LIN {X 0,Y 495.75,Z 552.238,A -85,B 0,C 180,E1 16037.936,E2 16037.936} C_VEL
LIN {X 0,Y 490.414,Z 542.078,A -85,B 0,C 180,E1 16035.4,E2 16035.4} C_VEL
LIN {X 0,Y 486.83,Z 535.501,A -85,B 0,C 180,E1 16033.42,E2 16033.42} C_VEL
LIN {X 0,Y 483.427,Z 530.223,A -85,B 0,C 180,E1 16031.272,E2 16031.272} C_VEL
LIN {X 0,Y 481.027,Z 526.46,A -85,B 0,C 180,E1 16029.452,E2 16029.452} C_VEL
LIN {X 0,Y 478.245,Z 521.895,A -85,B 0,C 180,E1 16026.724,E2 16026.724} C_VEL
LIN {X 0,Y 475.904,Z 518.407,A -85,B 0,C 180,E1 16023.011,E2 16023.011} C_VEL
LIN {X 0,Y 475.553,Z 516.68,A -85,B 0,C 180,E1 16021.446,E2 16021.446} C_VEL
LIN {X 0,Y 475.613,Z 516.934,A -85,B 0,C 180,E1 16017.711,E2 16017.711} C_VEL
LIN {X 0,Y 477.41,Z 521.143,A -85,B 0,C 180,E1 16013.748,E2 16013.748} C_VEL
LIN {X 0,Y 478.53,Z 522.413,A -85,B 0,C 180,E1 16012.436,E2 16012.436} C_VEL
LIN {X 0,Y 481.805,Z 527.661,A -85,B 0,C 180,E1 16009.417,E2 16009.417} C_VEL
LIN {X 0,Y 485.153,Z 532.978,A -85,B 0,C 180,E1 16007.078,E2 16007.078} C_VEL
LIN {X 0,Y 488.531,Z 538.287,A -85,B 0,C 180,E1 16005.116,E2 16005.116} C_VEL
LIN {X 0,Y 494.078,Z 547.334,A -85,B 0,C 180,E1 16002.389,E2 16002.389} C_VEL
LIN {X 0,Y 495.655,Z 550.313,A -85,B 0,C 180,E1 16001.678,E2 16001.678} C_VEL
LIN {X 0,Y 477.005,Z 773.14,A -85,B 0,C 180,E1 15998.26,E2 15998.26} C_VEL
LIN {X 0,Y 473.208,Z 814.507,A -85,B 0,C 180,E1 15997.599,E2 15997.599} C_VEL
LIN {X 0,Y 469.106,Z 841.171,A -85,B 0,C 180,E1 15997.058,E2 15997.058} C_VEL
LIN {X 0,Y 464.96,Z 862.529,A -85,B 0,C 180,E1 15996.503,E2 15996.503} C_VEL
LIN {X 0,Y 460.196,Z 883.041,A -85,B 0,C 180,E1 15995.856,E2 15995.856} C_VEL
LIN {X 0,Y 454.375,Z 904.584,A -85,B 0,C 180,E1 15995.041,E2 15995.041} C_VEL
LIN {X 0,Y 446.157,Z 930.766,A -85,B 0,C 180,E1 15993.836,E2 15993.836} C_VEL
LIN {X 0,Y 438.115,Z 952.919,A -85,B 0,C 180,E1 15992.594,E2 15992.594} C_VEL
LIN {X 0,Y 430.587,Z 971.671,A -85,B 0,C 180,E1 15991.371,E2 15991.371} C_VEL
LIN {X 0,Y 422.617,Z 989.978,A -85,B 0,C 180,E1 15989.986,E2 15989.986} C_VEL
LIN {X 0,Y 414.059,Z 1008.193,A -85,B 0,C 180,E1 15988.397,E2 15988.397} C_VEL
LIN {X 0,Y 402.823,Z 1030.327,A -85,B 0,C 180,E1 15986.126,E2 15986.126} C_VEL
LIN {X 0,Y 392.874,Z 1048.447,A -85,B 0,C 180,E1 15983.904,E2 15983.904} C_VEL
LIN {X 0,Y 384.294,Z 1063.355,A -85,B 0,C 180,E1 15981.789,E2 15981.789} C_VEL
LIN {X 0,Y 375.957,Z 1077.309,A -85,B 0,C 180,E1 15979.518,E2 15979.518} C_VEL
LIN {X 0,Y 367.251,Z 1091.49,A -85,B 0,C 180,E1 15976.856,E2 15976.856} C_VEL
LIN {X 0,Y 357.211,Z 1107.595,A -85,B 0,C 180,E1 15973.296,E2 15973.296} C_VEL
LIN {X 0,Y 348.718,Z 1120.908,A -85,B 0,C 180,E1 15969.747,E2 15969.747} C_VEL
LIN {X 0,Y 342.021,Z 1131.618,A -85,B 0,C 180,E1 15966.402,E2 15966.402} C_VEL
LIN {X 0,Y 336.338,Z 1141.067,A -85,B 0,C 180,E1 15962.957,E2 15962.957} C_VEL
LIN {X 0,Y 330.571,Z 1151.31,A -85,B 0,C 180,E1 15958.548,E2 15958.548} C_VEL
LIN {X 0,Y 326.088,Z 1159.977,A -85,B 0,C 180,E1 15953.875,E2 15953.875} C_VEL
LIN {X 0,Y 323.408,Z 1166.015,A -85,B 0,C 180,E1 15949.882,E2 15949.882} C_VEL
LIN {X 0,Y 321.713,Z 1170.693,A -85,B 0,C 180,E1 15946.058,E2 15946.058} C_VEL
LIN {X 0,Y 320.731,Z 1174.188,A -85,B 0,C 180,E1 15942.422,E2 15942.422} C_VEL
LIN {X 0,Y 320.245,Z 1176.775,A -85,B 0,C 180,E1 15938.8,E2 15938.8} C_VEL
LIN {X 0,Y 320.04,Z 1178.413,A -85,B 0,C 180,E1 15935.378,E2 15935.378} C_VEL
LIN {X 0,Y 319.982,Z 1179.268,A -85,B 0,C 180,E1 15931.97,E2 15931.97} C_VEL
LIN {X 0,Y 319.983,Z 1179.345,A -85,B 0,C 180,E1 15928.568,E2 15928.568} C_VEL
LIN {X 0,Y 320.024,Z 1178.581,A -85,B 0,C 180,E1 15924.981,E2 15924.981} C_VEL
LIN {X 0,Y 320.225,Z 1176.946,A -85,B 0,C 180,E1 15921.38,E2 15921.38} C_VEL
LIN {X 0,Y 320.681,Z 1174.428,A -85,B 0,C 180,E1 15917.759,E2 15917.759} C_VEL
LIN {X 0,Y 321.622,Z 1171.003,A -85,B 0,C 180,E1 15914.123,E2 15914.123} C_VEL
LIN {X 0,Y 323.269,Z 1166.396,A -85,B 0,C 180,E1 15910.298,E2 15910.298} C_VEL
LIN {X 0,Y 325.73,Z 1160.725,A -85,B 0,C 180,E1 15906.481,E2 15906.481} C_VEL
LIN {X 0,Y 329.298,Z 1153.603,A -85,B 0,C 180,E1 15902.515,E2 15902.515} C_VEL
LIN {X 0,Y 335.203,Z 1143.09,A -85,B 0,C 180,E1 15897.729,E2 15897.729} C_VEL
LIN {X 0,Y 341.588,Z 1132.376,A -85,B 0,C 180,E1 15893.753,E2 15893.753} C_VEL
LIN {X 0,Y 348.208,Z 1121.753,A -85,B 0,C 180,E1 15890.398,E2 15890.398} C_VEL
LIN {X 0,Y 355.813,Z 1109.777,A -85,B 0,C 180,E1 15887.154,E2 15887.154} C_VEL
LIN {X 0,Y 366.624,Z 1092.626,A -85,B 0,C 180,E1 15883.268,E2 15883.268} C_VEL
LIN {X 0,Y 372.671,Z 1082.974,A -85,B 0,C 180,E1 15881.378,E2 15881.378} C_VEL
LIN {X 0,Y 374.707,Z 1078.514,A -85,B 0,C 180,E1 15880.457,E2 15880.457} C_VEL
LIN {X 0,Y 377.403,Z 1067.82,A -85,B 0,C 180,E1 15877.896,E2 15877.896} C_VEL
LIN {X 0,Y 379.662,Z 1063.03,A -85,B 0,C 180,E1 15877.03,E2 15877.03} C_VEL
LIN {X 0,Y 390.229,Z 1045.195,A -85,B 0,C 180,E1 15874.537,E2 15874.537} C_VEL
LIN {X 0,Y 401.817,Z 1024.144,A -85,B 0,C 180,E1 15872.083,E2 15872.083} C_VEL
LIN {X 0,Y 411.116,Z 1006.054,A -85,B 0,C 180,E1 15870.302,E2 15870.302} C_VEL
LIN {X 0,Y 419.413,Z 988.742,A -85,B 0,C 180,E1 15868.825,E2 15868.825} C_VEL
LIN {X 0,Y 427.593,Z 970.262,A -85,B 0,C 180,E1 15867.452,E2 15867.452} C_VEL
LIN {X 0,Y 437.088,Z 946.84,A -85,B 0,C 180,E1 15865.973,E2 15865.973} C_VEL
LIN {X 0,Y 445.714,Z 922.226,A -85,B 0,C 180,E1 15864.698,E2 15864.698} C_VEL
LIN {X 0,Y 451.949,Z 902.144,A -85,B 0,C 180,E1 15863.824,E2 15863.824} C_VEL
LIN {X 0,Y 457.53,Z 881.65,A -85,B 0,C 180,E1 15863.07,E2 15863.07} C_VEL
LIN {X 0,Y 462.528,Z 860.189,A -85,B 0,C 180,E1 15862.411,E2 15862.411} C_VEL
LIN {X 0,Y 467.655,Z 833.351,A -85,B 0,C 180,E1 15861.757,E2 15861.757} C_VEL
LIN {X 0,Y 471.236,Z 806.582,A -85,B 0,C 180,E1 15861.267,E2 15861.267} C_VEL
LIN {X 0,Y 483.431,Z 664.825,A -85,B 0,C 180,E1 15859.081,E2 15859.081} C_VEL
LIN {X 0,Y 492.923,Z 555.55,A -85,B 0,C 180,E1 15857.416,E2 15857.416} C_VEL
LIN {X 0,Y 487.652,Z 546.708,A -85,B 0,C 180,E1 15854.79,E2 15854.79} C_VEL
LIN {X 0,Y 484.383,Z 541.518,A -85,B 0,C 180,E1 15852.882,E2 15852.882} C_VEL
LIN {X 0,Y 482.213,Z 538.052,A -85,B 0,C 180,E1 15851.421,E2 15851.421} C_VEL
LIN {X 0,Y 479.901,Z 534.242,A -85,B 0,C 180,E1 15849.595,E2 15849.595} C_VEL
LIN {X 0,Y 477.233,Z 529.795,A -85,B 0,C 180,E1 15846.859,E2 15846.859} C_VEL
LIN {X 0,Y 474.881,Z 525.658,A -85,B 0,C 180,E1 15842.414,E2 15842.414} C_VEL
LIN {X 0,Y 474.762,Z 524.669,A -85,B 0,C 180,E1 15841.448,E2 15841.448} C_VEL
LIN {X 0,Y 474.801,Z 524.83,A -85,B 0,C 180,E1 15838.673,E2 15838.673} C_VEL
LIN {X 0,Y 476.414,Z 529.01,A -85,B 0,C 180,E1 15834.581,E2 15834.581} C_VEL
LIN {X 0,Y 477.632,Z 530.406,A -85,B 0,C 180,E1 15833.086,E2 15833.086} C_VEL
LIN {X 0,Y 480.894,Z 535.8,A -85,B 0,C 180,E1 15830.002,E2 15830.002} C_VEL
LIN {X 0,Y 483.748,Z 540.41,A -85,B 0,C 180,E1 15827.95,E2 15827.95} C_VEL
LIN {X 0,Y 486.694,Z 545.279,A -85,B 0,C 180,E1 15826.152,E2 15826.152} C_VEL
LIN {X 0,Y 492.309,Z 556.092,A -85,B 0,C 180,E1 15823.207,E2 15823.207} C_VEL
LIN {X 0,Y 492.992,Z 557.773,A -85,B 0,C 180,E1 15822.869,E2 15822.869} C_VEL
LIN {X 0,Y 474.136,Z 778.593,A -85,B 0,C 180,E1 15819.49,E2 15819.49} C_VEL
LIN {X 0,Y 469.97,Z 824.297,A -85,B 0,C 180,E1 15818.766,E2 15818.766} C_VEL
LIN {X 0,Y 465.648,Z 852.231,A -85,B 0,C 180,E1 15818.23,E2 15818.23} C_VEL
LIN {X 0,Y 461.221,Z 874.106,A -85,B 0,C 180,E1 15817.714,E2 15817.714} C_VEL
LIN {X 0,Y 456.149,Z 895.17,A -85,B 0,C 180,E1 15817.097,E2 15817.097} C_VEL
LIN {X 0,Y 449.874,Z 917.56,A -85,B 0,C 180,E1 15816.302,E2 15816.302} C_VEL
LIN {X 0,Y 440.941,Z 944.901,A -85,B 0,C 180,E1 15815.096,E2 15815.096} C_VEL
LIN {X 0,Y 432.943,Z 966.301,A -85,B 0,C 180,E1 15813.945,E2 15813.945} C_VEL
LIN {X 0,Y 425.158,Z 985.312,A -85,B 0,C 180,E1 15812.742,E2 15812.742} C_VEL
LIN {X 0,Y 416.857,Z 1003.907,A -85,B 0,C 180,E1 15811.387,E2 15811.387} C_VEL
LIN {X 0,Y 406.65,Z 1025.184,A -85,B 0,C 180,E1 15809.567,E2 15809.567} C_VEL
LIN {X 0,Y 394.948,Z 1047.489,A -85,B 0,C 180,E1 15807.268,E2 15807.268} C_VEL
LIN {X 0,Y 385.523,Z 1064.419,A -85,B 0,C 180,E1 15805.208,E2 15805.208} C_VEL
LIN {X 0,Y 376.324,Z 1080.251,A -85,B 0,C 180,E1 15802.977,E2 15802.977} C_VEL
LIN {X 0,Y 366.484,Z 1096.63,A -85,B 0,C 180,E1 15800.297,E2 15800.297} C_VEL
LIN {X 0,Y 355.351,Z 1114.595,A -85,B 0,C 180,E1 15796.782,E2 15796.782} C_VEL
LIN {X 0,Y 346.694,Z 1128.363,A -85,B 0,C 180,E1 15793.572,E2 15793.572} C_VEL
LIN {X 0,Y 339.406,Z 1140.072,A -85,B 0,C 180,E1 15790.398,E2 15790.398} C_VEL
LIN {X 0,Y 332.394,Z 1151.594,A -85,B 0,C 180,E1 15786.77,E2 15786.77} C_VEL
LIN {X 0,Y 324.831,Z 1164.761,A -85,B 0,C 180,E1 15781.759,E2 15781.759} C_VEL
LIN {X 0,Y 320.263,Z 1173.478,A -85,B 0,C 180,E1 15777.722,E2 15777.722} C_VEL
LIN {X 0,Y 316.98,Z 1180.584,A -85,B 0,C 180,E1 15773.813,E2 15773.813} C_VEL
LIN {X 0,Y 314.614,Z 1186.622,A -85,B 0,C 180,E1 15769.824,E2 15769.824} C_VEL
LIN {X 0,Y 312.967,Z 1192.261,A -85,B 0,C 180,E1 15765.187,E2 15765.187} C_VEL
LIN {X 0,Y 312.171,Z 1196.482,A -85,B 0,C 180,E1 15760.333,E2 15760.333} C_VEL
LIN {X 0,Y 311.987,Z 1198.799,A -85,B 0,C 180,E1 15756.256,E2 15756.256} C_VEL
LIN {X 0,Y 311.979,Z 1199.933,A -85,B 0,C 180,E1 15752.572,E2 15752.572} C_VEL
LIN {X 0,Y 311.983,Z 1200.121,A -85,B 0,C 180,E1 15748.898,E2 15748.898} C_VEL
LIN {X 0,Y 311.974,Z 1199.365,A -85,B 0,C 180,E1 15745.22,E2 15745.22} C_VEL
LIN {X 0,Y 312.051,Z 1197.662,A -85,B 0,C 180,E1 15741.524,E2 15741.524} C_VEL
LIN {X 0,Y 312.398,Z 1194.842,A -85,B 0,C 180,E1 15737.617,E2 15737.617} C_VEL
LIN {X 0,Y 313.276,Z 1190.964,A -85,B 0,C 180,E1 15733.688,E2 15733.688} C_VEL
LIN {X 0,Y 314.826,Z 1186.005,A -85,B 0,C 180,E1 15729.747,E2 15729.747} C_VEL
LIN {X 0,Y 317.113,Z 1180.25,A -85,B 0,C 180,E1 15726,E2 15726} C_VEL
LIN {X 0,Y 320.564,Z 1172.85,A -85,B 0,C 180,E1 15721.973,E2 15721.973} C_VEL
LIN {X 0,Y 326.29,Z 1162.177,A -85,B 0,C 180,E1 15717.154,E2 15717.154} C_VEL
LIN {X 0,Y 333.014,Z 1150.506,A -85,B 0,C 180,E1 15712.88,E2 15712.88} C_VEL
LIN {X 0,Y 339.761,Z 1139.443,A -85,B 0,C 180,E1 15709.431,E2 15709.431} C_VEL
LIN {X 0,Y 347.501,Z 1127.012,A -85,B 0,C 180,E1 15706.098,E2 15706.098} C_VEL
LIN {X 0,Y 358.082,Z 1110.175,A -85,B 0,C 180,E1 15702.296,E2 15702.296} C_VEL
LIN {X 0,Y 368.02,Z 1093.965,A -85,B 0,C 180,E1 15699.258,E2 15699.258} C_VEL
LIN {X 0,Y 377.147,Z 1078.74,A -85,B 0,C 180,E1 15696.81,E2 15696.81} C_VEL
LIN {X 0,Y 386.604,Z 1062.403,A -85,B 0,C 180,E1 15694.541,E2 15694.541} C_VEL
LIN {X 0,Y 398.513,Z 1040.77,A -85,B 0,C 180,E1 15692.002,E2 15692.002} C_VEL
LIN {X 0,Y 408.806,Z 1020.52,A -85,B 0,C 180,E1 15690.025,E2 15690.025} C_VEL
LIN {X 0,Y 417.516,Z 1002.219,A -85,B 0,C 180,E1 15688.492,E2 15688.492} C_VEL
LIN {X 0,Y 425.839,Z 983.449,A -85,B 0,C 180,E1 15687.142,E2 15687.142} C_VEL
LIN {X 0,Y 434.731,Z 961.518,A -85,B 0,C 180,E1 15685.786,E2 15685.786} C_VEL
LIN {X 0,Y 443.915,Z 935.872,A -85,B 0,C 180,E1 15684.485,E2 15684.485} C_VEL
LIN {X 0,Y 450.606,Z 914.601,A -85,B 0,C 180,E1 15683.593,E2 15683.593} C_VEL
LIN {X 0,Y 456.321,Z 893.984,A -85,B 0,C 180,E1 15682.873,E2 15682.873} C_VEL
LIN {X 0,Y 461.332,Z 872.995,A -85,B 0,C 180,E1 15682.264,E2 15682.264} C_VEL
LIN {X 0,Y 466.121,Z 848.981,A -85,B 0,C 180,E1 15681.709,E2 15681.709} C_VEL
LIN {X 0,Y 470.294,Z 819.745,A -85,B 0,C 180,E1 15681.166,E2 15681.166} C_VEL
LIN {X 0,Y 476.185,Z 752.192,A -85,B 0,C 180,E1 15680.11,E2 15680.11} C_VEL
LIN {X 0,Y 492.837,Z 557.39,A -85,B 0,C 180,E1 15677.124,E2 15677.124} C_VEL
LIN {X 0,Y 487.943,Z 547.91,A -85,B 0,C 180,E1 15674.66,E2 15674.66} C_VEL
LIN {X 0,Y 485.144,Z 542.775,A -85,B 0,C 180,E1 15673.043,E2 15673.043} C_VEL
LIN {X 0,Y 482.105,Z 537.911,A -85,B 0,C 180,E1 15671.061,E2 15671.061} C_VEL
LIN {X 0,Y 479.904,Z 534.344,A -85,B 0,C 180,E1 15669.353,E2 15669.353} C_VEL
LIN {X 0,Y 477.055,Z 529.687,A -85,B 0,C 180,E1 15666.499,E2 15666.499} C_VEL
LIN {X 0,Y 474.846,Z 526.136,A -85,B 0,C 180,E1 15662.776,E2 15662.776} C_VEL
LIN {X 0,Y 474.55,Z 524.614,A -85,B 0,C 180,E1 15661.328,E2 15661.328} C_VEL
LIN {X 0,Y 474.611,Z 524.819,A -85,B 0,C 180,E1 15657.827,E2 15657.827} C_VEL
LIN {X 0,Y 476.436,Z 529.122,A -85,B 0,C 180,E1 15653.735,E2 15653.735} C_VEL
LIN {X 0,Y 477.439,Z 530.341,A -85,B 0,C 180,E1 15652.539,E2 15652.539} C_VEL
LIN {X 0,Y 480.592,Z 535.493,A -85,B 0,C 180,E1 15649.572,E2 15649.572} C_VEL
LIN {X 0,Y 483.792,Z 540.671,A -85,B 0,C 180,E1 15647.287,E2 15647.287} C_VEL
LIN {X 0,Y 487.114,Z 545.999,A -85,B 0,C 180,E1 15645.315,E2 15645.315} C_VEL
LIN {X 0,Y 492.64,Z 555.185,A -85,B 0,C 180,E1 15642.549,E2 15642.549} C_VEL
LIN {X 0,Y 492.74,Z 555.792,A -85,B 0,C 180,E1 15642.482,E2 15642.482} C_VEL
LIN {X 0,Y 473.681,Z 778.427,A -85,B 0,C 180,E1 15639.082,E2 15639.082} C_VEL
LIN {X 0,Y 470.001,Z 816.245,A -85,B 0,C 180,E1 15638.474,E2 15638.474} C_VEL
LIN {X 0,Y 465.993,Z 841.708,A -85,B 0,C 180,E1 15637.959,E2 15637.959} C_VEL
LIN {X 0,Y 461.747,Z 863.128,A -85,B 0,C 180,E1 15637.408,E2 15637.408} C_VEL
LIN {X 0,Y 456.779,Z 884.051,A -85,B 0,C 180,E1 15636.751,E2 15636.751} C_VEL
LIN {X 0,Y 450.303,Z 907.411,A -85,B 0,C 180,E1 15635.865,E2 15635.865} C_VEL
LIN {X 0,Y 441.922,Z 933.032,A -85,B 0,C 180,E1 15634.672,E2 15634.672} C_VEL
LIN {X 0,Y 434.435,Z 953.191,A -85,B 0,C 180,E1 15633.545,E2 15633.545} C_VEL
LIN {X 0,Y 426.746,Z 971.943,A -85,B 0,C 180,E1 15632.331,E2 15632.331} C_VEL
LIN {X 0,Y 418.595,Z 990.251,A -85,B 0,C 180,E1 15630.954,E2 15630.954} C_VEL
LIN {X 0,Y 410.011,Z 1008.079,A -85,B 0,C 180,E1 15629.41,E2 15629.41} C_VEL
LIN {X 0,Y 398.607,Z 1030.052,A -85,B 0,C 180,E1 15627.172,E2 15627.172} C_VEL
LIN {X 0,Y 388.064,Z 1048.722,A -85,B 0,C 180,E1 15624.89,E2 15624.89} C_VEL
LIN {X 0,Y 379.22,Z 1063.631,A -85,B 0,C 180,E1 15622.774,E2 15622.774} C_VEL
LIN {X 0,Y 370.328,Z 1078.042,A -85,B 0,C 180,E1 15620.416,E2 15620.416} C_VEL
LIN {X 0,Y 360.658,Z 1093.281,A -85,B 0,C 180,E1 15617.513,E2 15617.513} C_VEL
LIN {X 0,Y 349.663,Z 1110.098,A -85,B 0,C 180,E1 15613.658,E2 15613.658} C_VEL
LIN {X 0,Y 341.598,Z 1122.307,A -85,B 0,C 180,E1 15610.306,E2 15610.306} C_VEL
LIN {X 0,Y 334.698,Z 1132.9,A -85,B 0,C 180,E1 15606.902,E2 15606.902} C_VEL
LIN {X 0,Y 327.717,Z 1144.13,A -85,B 0,C 180,E1 15602.637,E2 15602.637} C_VEL
LIN {X 0,Y 321.842,Z 1154.033,A -85,B 0,C 180,E1 15597.976,E2 15597.976} C_VEL
LIN {X 0,Y 318.242,Z 1160.836,A -85,B 0,C 180,E1 15594.107,E2 15594.107} C_VEL
LIN {X 0,Y 315.58,Z 1166.532,A -85,B 0,C 180,E1 15590.203,E2 15590.203} C_VEL
LIN {X 0,Y 313.8,Z 1171.161,A -85,B 0,C 180,E1 15586.284,E2 15586.284} C_VEL
LIN {X 0,Y 312.73,Z 1174.763,A -85,B 0,C 180,E1 15582.369,E2 15582.369} C_VEL
LIN {X 0,Y 312.206,Z 1177.493,A -85,B 0,C 180,E1 15578.259,E2 15578.259} C_VEL
LIN {X 0,Y 312.01,Z 1179.329,A -85,B 0,C 180,E1 15573.675,E2 15573.675} C_VEL
LIN {X 0,Y 311.98,Z 1179.696,A -85,B 0,C 180,E1 15569.265,E2 15569.265} C_VEL
LIN {X 0,Y 312.026,Z 1178.975,A -85,B 0,C 180,E1 15565.221,E2 15565.221} C_VEL
LIN {X 0,Y 312.237,Z 1177.32,A -85,B 0,C 180,E1 15561.344,E2 15561.344} C_VEL
LIN {X 0,Y 312.753,Z 1174.694,A -85,B 0,C 180,E1 15557.444,E2 15557.444} C_VEL
LIN {X 0,Y 313.767,Z 1171.27,A -85,B 0,C 180,E1 15553.715,E2 15553.715} C_VEL
LIN {X 0,Y 315.537,Z 1166.665,A -85,B 0,C 180,E1 15549.794,E2 15549.794} C_VEL
LIN {X 0,Y 318.173,Z 1160.995,A -85,B 0,C 180,E1 15545.888,E2 15545.888} C_VEL
LIN {X 0,Y 321.955,Z 1153.874,A -85,B 0,C 180,E1 15541.833,E2 15541.833} C_VEL
LIN {X 0,Y 328.29,Z 1143.195,A -85,B 0,C 180,E1 15536.886,E2 15536.886} C_VEL
LIN {X 0,Y 334.888,Z 1132.649,A -85,B 0,C 180,E1 15532.908,E2 15532.908} C_VEL
LIN {X 0,Y 341.823,Z 1122.024,A -85,B 0,C 180,E1 15529.506,E2 15529.506} C_VEL
LIN {X 0,Y 349.747,Z 1110.049,A -85,B 0,C 180,E1 15526.225,E2 15526.225} C_VEL
LIN {X 0,Y 360.963,Z 1092.897,A -85,B 0,C 180,E1 15522.304,E2 15522.304} C_VEL
LIN {X 0,Y 369.922,Z 1078.822,A -85,B 0,C 180,E1 15519.617,E2 15519.617} C_VEL
LIN {X 0,Y 379.214,Z 1063.772,A -85,B 0,C 180,E1 15517.144,E2 15517.144} C_VEL
LIN {X 0,Y 379.662,Z 1063.03,A -85,B 0,C 180,E1 15517.03,E2 15517.03} C_VEL
LIN {X 0,Y 381.998,Z 1058.28,A -85,B 0,C 180,E1 15516.179,E2 15516.179} C_VEL
LIN {X 0,Y 385.839,Z 1045.871,A -85,B 0,C 180,E1 15513.666,E2 15513.666} C_VEL
LIN {X 0,Y 387.983,Z 1041.376,A -85,B 0,C 180,E1 15513.013,E2 15513.013} C_VEL
LIN {X 0,Y 398.472,Z 1022.606,A -85,B 0,C 180,E1 15510.89,E2 15510.89} C_VEL
LIN {X 0,Y 407.704,Z 1004.997,A -85,B 0,C 180,E1 15509.184,E2 15509.184} C_VEL
LIN {X 0,Y 416.575,Z 986.821,A -85,B 0,C 180,E1 15507.667,E2 15507.667} C_VEL
LIN {X 0,Y 426.775,Z 964.068,A -85,B 0,C 180,E1 15506.042,E2 15506.042} C_VEL
LIN {X 0,Y 436.132,Z 940.161,A -85,B 0,C 180,E1 15504.633,E2 15504.633} C_VEL
LIN {X 0,Y 443.139,Z 920.237,A -85,B 0,C 180,E1 15503.643,E2 15503.643} C_VEL
LIN {X 0,Y 449.394,Z 900.233,A -85,B 0,C 180,E1 15502.797,E2 15502.797} C_VEL
LIN {X 0,Y 455.202,Z 878.959,A -85,B 0,C 180,E1 15502.039,E2 15502.039} C_VEL
LIN {X 0,Y 461.406,Z 851.698,A -85,B 0,C 180,E1 15501.254,E2 15501.254} C_VEL
LIN {X 0,Y 465.764,Z 826.637,A -85,B 0,C 180,E1 15500.703,E2 15500.703} C_VEL
LIN {X 0,Y 468.659,Z 804.306,A -85,B 0,C 180,E1 15500.313,E2 15500.313} C_VEL
LIN {X 0,Y 487.612,Z 588.987,A -85,B 0,C 180,E1 15497.027,E2 15497.027} C_VEL
LIN {X 0,Y 490.092,Z 561.078,A -85,B 0,C 180,E1 15496.597,E2 15496.597} C_VEL
LIN {X 0,Y 485.316,Z 552.927,A -85,B 0,C 180,E1 15494.07,E2 15494.07} C_VEL
LIN {X 0,Y 481.315,Z 546.322,A -85,B 0,C 180,E1 15491.504,E2 15491.504} C_VEL
LIN {X 0,Y 478.644,Z 541.962,A -85,B 0,C 180,E1 15489.378,E2 15489.378} C_VEL
LIN {X 0,Y 476.054,Z 537.597,A -85,B 0,C 180,E1 15486.634,E2 15486.634} C_VEL
LIN {X 0,Y 473.877,Z 533.539,A -85,B 0,C 180,E1 15482.298,E2 15482.298} C_VEL
LIN {X 0,Y 473.767,Z 532.606,A -85,B 0,C 180,E1 15481.33,E2 15481.33} C_VEL
LIN {X 0,Y 473.816,Z 532.859,A -85,B 0,C 180,E1 15478.67,E2 15478.67} C_VEL
LIN {X 0,Y 475.44,Z 536.983,A -85,B 0,C 180,E1 15474.569,E2 15474.569} C_VEL
LIN {X 0,Y 476.543,Z 538.33,A -85,B 0,C 180,E1 15473.192,E2 15473.192} C_VEL
LIN {X 0,Y 479.684,Z 543.623,A -85,B 0,C 180,E1 15470.158,E2 15470.158} C_VEL
LIN {X 0,Y 482.402,Z 548.108,A -85,B 0,C 180,E1 15468.159,E2 15468.159} C_VEL
LIN {X 0,Y 485.142,Z 552.741,A -85,B 0,C 180,E1 15466.441,E2 15466.441} C_VEL
LIN {X 0,Y 490.207,Z 562.772,A -85,B 0,C 180,E1 15463.689,E2 15463.689} C_VEL
LIN {X 0,Y 470.968,Z 783.121,A -85,B 0,C 180,E1 15460.334,E2 15460.334} C_VEL
LIN {X 0,Y 466.929,Z 825.661,A -85,B 0,C 180,E1 15459.659,E2 15459.659} C_VEL
LIN {X 0,Y 462.572,Z 852.763,A -85,B 0,C 180,E1 15459.139,E2 15459.139} C_VEL
LIN {X 0,Y 458.062,Z 874.554,A -85,B 0,C 180,E1 15458.63,E2 15458.63} C_VEL
LIN {X 0,Y 452.866,Z 895.656,A -85,B 0,C 180,E1 15458.016,E2 15458.016} C_VEL
LIN {X 0,Y 446.126,Z 919.148,A -85,B 0,C 180,E1 15457.186,E2 15457.186} C_VEL
LIN {X 0,Y 437.217,Z 945.579,A -85,B 0,C 180,E1 15456.019,E2 15456.019} C_VEL
LIN {X 0,Y 429.38,Z 966.099,A -85,B 0,C 180,E1 15454.924,E2 15454.924} C_VEL
LIN {X 0,Y 421.451,Z 985.047,A -85,B 0,C 180,E1 15453.737,E2 15453.737} C_VEL
LIN {X 0,Y 412.962,Z 1003.64,A -85,B 0,C 180,E1 15452.394,E2 15452.394} C_VEL
LIN {X 0,Y 402.393,Z 1025.151,A -85,B 0,C 180,E1 15450.565,E2 15450.565} C_VEL
LIN {X 0,Y 390.855,Z 1046.591,A -85,B 0,C 180,E1 15448.37,E2 15448.37} C_VEL
LIN {X 0,Y 381.022,Z 1063.788,A -85,B 0,C 180,E1 15446.29,E2 15446.29} C_VEL
LIN {X 0,Y 371.62,Z 1079.509,A -85,B 0,C 180,E1 15444.081,E2 15444.081} C_VEL
LIN {X 0,Y 362.122,Z 1094.814,A -85,B 0,C 180,E1 15441.591,E2 15441.591} C_VEL
LIN {X 0,Y 350.571,Z 1112.894,A -85,B 0,C 180,E1 15438.107,E2 15438.107} C_VEL
LIN {X 0,Y 341.032,Z 1127.44,A -85,B 0,C 180,E1 15434.72,E2 15434.72} C_VEL
LIN {X 0,Y 333.377,Z 1139.21,A -85,B 0,C 180,E1 15431.515,E2 15431.515} C_VEL
LIN {X 0,Y 326.326,Z 1150.266,A -85,B 0,C 180,E1 15428.014,E2 15428.014} C_VEL
LIN {X 0,Y 318.979,Z 1162.397,A -85,B 0,C 180,E1 15423.482,E2 15423.482} C_VEL
LIN {X 0,Y 313.256,Z 1172.476,A -85,B 0,C 180,E1 15418.814,E2 15418.814} C_VEL
LIN {X 0,Y 309.654,Z 1179.685,A -85,B 0,C 180,E1 15414.82,E2 15414.82} C_VEL
LIN {X 0,Y 307.077,Z 1185.75,A -85,B 0,C 180,E1 15410.788,E2 15410.788} C_VEL
LIN {X 0,Y 305.397,Z 1190.707,A -85,B 0,C 180,E1 15406.745,E2 15406.745} C_VEL
LIN {X 0,Y 304.444,Z 1194.585,A -85,B 0,C 180,E1 15402.711,E2 15402.711} C_VEL
LIN {X 0,Y 304.053,Z 1197.522,A -85,B 0,C 180,E1 15398.51,E2 15398.51} C_VEL
LIN {X 0,Y 303.972,Z 1199.458,A -85,B 0,C 180,E1 15393.961,E2 15393.961} C_VEL
LIN {X 0,Y 303.981,Z 1199.951,A -85,B 0,C 180,E1 15389.623,E2 15389.623} C_VEL
LIN {X 0,Y 303.976,Z 1199.19,A -85,B 0,C 180,E1 15385.333,E2 15385.333} C_VEL
LIN {X 0,Y 304.061,Z 1197.396,A -85,B 0,C 180,E1 15381.3,E2 15381.3} C_VEL
LIN {X 0,Y 304.447,Z 1194.562,A -85,B 0,C 180,E1 15377.275,E2 15377.275} C_VEL
LIN {X 0,Y 305.397,Z 1190.694,A -85,B 0,C 180,E1 15373.255,E2 15373.255} C_VEL
LIN {X 0,Y 307.076,Z 1185.733,A -85,B 0,C 180,E1 15369.212,E2 15369.212} C_VEL
LIN {X 0,Y 309.513,Z 1179.976,A -85,B 0,C 180,E1 15365.372,E2 15365.372} C_VEL
LIN {X 0,Y 313.059,Z 1172.811,A -85,B 0,C 180,E1 15361.375,E2 15361.375} C_VEL
LIN {X 0,Y 318.719,Z 1162.79,A -85,B 0,C 180,E1 15356.702,E2 15356.702} C_VEL
LIN {X 0,Y 325.996,Z 1150.754,A -85,B 0,C 180,E1 15352.163,E2 15352.163} C_VEL
LIN {X 0,Y 333.027,Z 1139.704,A -85,B 0,C 180,E1 15348.643,E2 15348.643} C_VEL
LIN {X 0,Y 341.025,Z 1127.381,A -85,B 0,C 180,E1 15345.279,E2 15345.279} C_VEL
LIN {X 0,Y 351.534,Z 1111.382,A -85,B 0,C 180,E1 15341.579,E2 15341.579} C_VEL
LIN {X 0,Y 362.218,Z 1094.545,A -85,B 0,C 180,E1 15338.377,E2 15338.377} C_VEL
LIN {X 0,Y 371.619,Z 1079.382,A -85,B 0,C 180,E1 15335.913,E2 15335.913} C_VEL
LIN {X 0,Y 381.009,Z 1063.665,A -85,B 0,C 180,E1 15333.708,E2 15333.708} C_VEL
LIN {X 0,Y 391.261,Z 1045.709,A -85,B 0,C 180,E1 15331.543,E2 15331.543} C_VEL
LIN {X 0,Y 403.555,Z 1022.582,A -85,B 0,C 180,E1 15329.216,E2 15329.216} C_VEL
LIN {X 0,Y 413.29,Z 1002.684,A -85,B 0,C 180,E1 15327.544,E2 15327.544} C_VEL
LIN {X 0,Y 421.789,Z 983.992,A -85,B 0,C 180,E1 15326.203,E2 15326.203} C_VEL
LIN {X 0,Y 430.122,Z 963.964,A -85,B 0,C 180,E1 15324.962,E2 15324.962} C_VEL
LIN {X 0,Y 439.809,Z 937.993,A -85,B 0,C 180,E1 15323.627,E2 15323.627} C_VEL
LIN {X 0,Y 447.035,Z 915.617,A -85,B 0,C 180,E1 15322.689,E2 15322.689} C_VEL
LIN {X 0,Y 453.04,Z 894.453,A -85,B 0,C 180,E1 15321.954,E2 15321.954} C_VEL
LIN {X 0,Y 458.199,Z 873.314,A -85,B 0,C 180,E1 15321.346,E2 15321.346} C_VEL
LIN {X 0,Y 462.877,Z 850.403,A -85,B 0,C 180,E1 15320.819,E2 15320.819} C_VEL
LIN {X 0,Y 467.407,Z 819.829,A -85,B 0,C 180,E1 15320.251,E2 15320.251} C_VEL
LIN {X 0,Y 473.074,Z 756.583,A -85,B 0,C 180,E1 15319.266,E2 15319.266} C_VEL
LIN {X 0,Y 490.037,Z 562.627,A -85,B 0,C 180,E1 15316.311,E2 15316.311} C_VEL
LIN {X 0,Y 484.634,Z 551.909,A -85,B 0,C 180,E1 15313.361,E2 15313.361} C_VEL
LIN {X 0,Y 480.872,Z 545.719,A -85,B 0,C 180,E1 15310.907,E2 15310.907} C_VEL
LIN {X 0,Y 478.639,Z 542.06,A -85,B 0,C 180,E1 15309.135,E2 15309.135} C_VEL
LIN {X 0,Y 475.977,Z 537.569,A -85,B 0,C 180,E1 15306.392,E2 15306.392} C_VEL
LIN {X 0,Y 473.828,Z 534.016,A -85,B 0,C 180,E1 15302.661,E2 15302.661} C_VEL
LIN {X 0,Y 473.549,Z 532.556,A -85,B 0,C 180,E1 15301.21,E2 15301.21} C_VEL
LIN {X 0,Y 473.611,Z 532.704,A -85,B 0,C 180,E1 15297.943,E2 15297.943} C_VEL
LIN {X 0,Y 475.371,Z 537.003,A -85,B 0,C 180,E1 15293.842,E2 15293.842} C_VEL
LIN {X 0,Y 476.302,Z 538.149,A -85,B 0,C 180,E1 15292.703,E2 15292.703} C_VEL
LIN {X 0,Y 479.313,Z 543.185,A -85,B 0,C 180,E1 15289.786,E2 15289.786} C_VEL
LIN {X 0,Y 482.445,Z 548.375,A -85,B 0,C 180,E1 15287.492,E2 15287.492} C_VEL
LIN {X 0,Y 485.806,Z 553.877,A -85,B 0,C 180,E1 15285.457,E2 15285.457} C_VEL
LIN {X 0,Y 489.94,Z 561.085,A -85,B 0,C 180,E1 15283.299,E2 15283.299} C_VEL
LIN {X 0,Y 470.368,Z 784.753,A -85,B 0,C 180,E1 15279.899,E2 15279.899} C_VEL
LIN {X 0,Y 466.59,Z 820.086,A -85,B 0,C 180,E1 15279.321,E2 15279.321} C_VEL
LIN {X 0,Y 462.848,Z 843.044,A -85,B 0,C 180,E1 15278.854,E2 15278.854} C_VEL
LIN {X 0,Y 458.532,Z 864.266,A -85,B 0,C 180,E1 15278.309,E2 15278.309} C_VEL
LIN {X 0,Y 453.285,Z 885.797,A -85,B 0,C 180,E1 15277.635,E2 15277.635} C_VEL
LIN {X 0,Y 445.951,Z 911.402,A -85,B 0,C 180,E1 15276.654,E2 15276.654} C_VEL
LIN {X 0,Y 437.783,Z 935.301,A -85,B 0,C 180,E1 15275.524,E2 15275.524} C_VEL
LIN {X 0,Y 430.519,Z 954.356,A -85,B 0,C 180,E1 15274.458,E2 15274.458} C_VEL
LIN {X 0,Y 422.675,Z 973.02,A -85,B 0,C 180,E1 15273.252,E2 15273.252} C_VEL
LIN {X 0,Y 414.006,Z 991.979,A -85,B 0,C 180,E1 15271.824,E2 15271.824} C_VEL
LIN {X 0,Y 403.269,Z 1013.62,A -85,B 0,C 180,E1 15269.917,E2 15269.917} C_VEL
LIN {X 0,Y 391.984,Z 1034.164,A -85,B 0,C 180,E1 15267.734,E2 15267.734} C_VEL
LIN {X 0,Y 382.771,Z 1049.997,A -85,B 0,C 180,E1 15265.766,E2 15265.766} C_VEL
LIN {X 0,Y 373.695,Z 1064.818,A -85,B 0,C 180,E1 15263.644,E2 15263.644} C_VEL
LIN {X 0,Y 364.318,Z 1079.525,A -85,B 0,C 180,E1 15261.208,E2 15261.208} C_VEL
LIN {X 0,Y 352.972,Z 1096.788,A -85,B 0,C 180,E1 15257.827,E2 15257.827} C_VEL
LIN {X 0,Y 343.059,Z 1111.261,A -85,B 0,C 180,E1 15254.386,E2 15254.386} C_VEL
LIN {X 0,Y 335.284,Z 1122.583,A -85,B 0,C 180,E1 15251.227,E2 15251.227} C_VEL
LIN {X 0,Y 328.064,Z 1133.176,A -85,B 0,C 180,E1 15247.778,E2 15247.778} C_VEL
LIN {X 0,Y 320.799,Z 1144.302,A -85,B 0,C 180,E1 15243.481,E2 15243.481} C_VEL
LIN {X 0,Y 314.512,Z 1154.348,A -85,B 0,C 180,E1 15238.663,E2 15238.663} C_VEL
LIN {X 0,Y 310.557,Z 1161.402,A -85,B 0,C 180,E1 15234.54,E2 15234.54} C_VEL
LIN {X 0,Y 307.763,Z 1167.049,A -85,B 0,C 180,E1 15230.54,E2 15230.54} C_VEL
LIN {X 0,Y 305.822,Z 1171.828,A -85,B 0,C 180,E1 15226.33,E2 15226.33} C_VEL
LIN {X 0,Y 304.575,Z 1176.102,A -85,B 0,C 180,E1 15221.36,E2 15221.36} C_VEL
LIN {X 0,Y 304.11,Z 1178.616,A -85,B 0,C 180,E1 15216.608,E2 15216.608} C_VEL
LIN {X 0,Y 303.996,Z 1179.729,A -85,B 0,C 180,E1 15212.639,E2 15212.639} C_VEL
LIN {X 0,Y 303.99,Z 1179.914,A -85,B 0,C 180,E1 15208.869,E2 15208.869} C_VEL
LIN {X 0,Y 304.038,Z 1179.172,A -85,B 0,C 180,E1 15204.906,E2 15204.906} C_VEL
LIN {X 0,Y 304.264,Z 1177.584,A -85,B 0,C 180,E1 15201.115,E2 15201.115} C_VEL
LIN {X 0,Y 304.832,Z 1174.96,A -85,B 0,C 180,E1 15197.112,E2 15197.112} C_VEL
LIN {X 0,Y 306.003,Z 1171.339,A -85,B 0,C 180,E1 15193.094,E2 15193.094} C_VEL
LIN {X 0,Y 307.943,Z 1166.688,A -85,B 0,C 180,E1 15189.074,E2 15189.074} C_VEL
LIN {X 0,Y 310.967,Z 1160.678,A -85,B 0,C 180,E1 15184.886,E2 15184.886} C_VEL
LIN {X 0,Y 315.974,Z 1152.066,A -85,B 0,C 180,E1 15180.002,E2 15180.002} C_VEL
LIN {X 0,Y 322.345,Z 1141.844,A -85,B 0,C 180,E1 15175.415,E2 15175.415} C_VEL
LIN {X 0,Y 328.61,Z 1132.417,A -85,B 0,C 180,E1 15171.854,E2 15171.854} C_VEL
LIN {X 0,Y 335.919,Z 1121.735,A -85,B 0,C 180,E1 15168.413,E2 15168.413} C_VEL
LIN {X 0,Y 345.539,Z 1107.83,A -85,B 0,C 180,E1 15164.616,E2 15164.616} C_VEL
LIN {X 0,Y 356.221,Z 1091.922,A -85,B 0,C 180,E1 15161.058,E2 15161.058} C_VEL
LIN {X 0,Y 365.456,Z 1077.871,A -85,B 0,C 180,E1 15158.395,E2 15158.395} C_VEL
LIN {X 0,Y 374.648,Z 1063.425,A -85,B 0,C 180,E1 15156.037,E2 15156.037} C_VEL
LIN {X 0,Y 385.298,Z 1045.963,A -85,B 0,C 180,E1 15153.592,E2 15153.592} C_VEL
LIN {X 0,Y 387.983,Z 1041.376,A -85,B 0,C 180,E1 15153.013,E2 15153.013} C_VEL
LIN {X 0,Y 390.415,Z 1036.172,A -85,B 0,C 180,E1 15152.257,E2 15152.257} C_VEL
LIN {X 0,Y 394.483,Z 1023.477,A -85,B 0,C 180,E1 15150.056,E2 15150.056} C_VEL
LIN {X 0,Y 397.09,Z 1017.894,A -85,B 0,C 180,E1 15149.36,E2 15149.36} C_VEL
LIN {X 0,Y 409.332,Z 994.364,A -85,B 0,C 180,E1 15147.236,E2 15147.236} C_VEL
LIN {X 0,Y 418.735,Z 974.355,A -85,B 0,C 180,E1 15145.727,E2 15145.727} C_VEL
LIN {X 0,Y 427.064,Z 955.007,A -85,B 0,C 180,E1 15144.482,E2 15144.482} C_VEL
LIN {X 0,Y 435.063,Z 934.431,A -85,B 0,C 180,E1 15143.347,E2 15143.347} C_VEL
LIN {X 0,Y 444.157,Z 907.765,A -85,B 0,C 180,E1 15142.129,E2 15142.129} C_VEL
LIN {X 0,Y 450.694,Z 885.104,A -85,B 0,C 180,E1 15141.289,E2 15141.289} C_VEL
LIN {X 0,Y 455.916,Z 863.935,A -85,B 0,C 180,E1 15140.639,E2 15140.639} C_VEL
LIN {X 0,Y 460.317,Z 842.558,A -85,B 0,C 180,E1 15140.1,E2 15140.1} C_VEL
LIN {X 0,Y 464.369,Z 817.817,A -85,B 0,C 180,E1 15139.609,E2 15139.609} C_VEL
LIN {X 0,Y 468.167,Z 781.28,A -85,B 0,C 180,E1 15139.026,E2 15139.026} C_VEL
LIN {X 0,Y 487.393,Z 566.593,A -85,B 0,C 180,E1 15135.78,E2 15135.78} C_VEL
LIN {X 0,Y 482.594,Z 558.318,A -85,B 0,C 180,E1 15133.052,E2 15133.052} C_VEL
LIN {X 0,Y 479.44,Z 553.194,A -85,B 0,C 180,E1 15130.879,E2 15130.879} C_VEL
LIN {X 0,Y 477.393,Z 549.681,A -85,B 0,C 180,E1 15129.159,E2 15129.159} C_VEL
LIN {X 0,Y 474.981,Z 545.482,A -85,B 0,C 180,E1 15126.527,E2 15126.527} C_VEL
LIN {X 0,Y 472.859,Z 541.27,A -85,B 0,C 180,E1 15122.06,E2 15122.06} C_VEL
LIN {X 0,Y 472.774,Z 540.543,A -85,B 0,C 180,E1 15121.212,E2 15121.212} C_VEL
LIN {X 0,Y 472.823,Z 540.738,A -85,B 0,C 180,E1 15118.788,E2 15118.788} C_VEL
LIN {X 0,Y 474.379,Z 544.866,A -85,B 0,C 180,E1 15114.679,E2 15114.679} C_VEL
LIN {X 0,Y 475.41,Z 546.136,A -85,B 0,C 180,E1 15113.357,E2 15113.357} C_VEL
LIN {X 0,Y 478.409,Z 551.311,A -85,B 0,C 180,E1 15110.375,E2 15110.375} C_VEL
LIN {X 0,Y 481.063,Z 555.806,A -85,B 0,C 180,E1 15108.369,E2 15108.369} C_VEL
LIN {X 0,Y 483.65,Z 560.304,A -85,B 0,C 180,E1 15106.703,E2 15106.703} C_VEL
LIN {X 0,Y 487.482,Z 568.227,A -85,B 0,C 180,E1 15104.512,E2 15104.512} C_VEL
LIN {X 0,Y 467.814,Z 788.68,A -85,B 0,C 180,E1 15101.174,E2 15101.174} C_VEL
LIN {X 0,Y 463.97,Z 826.883,A -85,B 0,C 180,E1 15100.564,E2 15100.564} C_VEL
LIN {X 0,Y 459.715,Z 852.773,A -85,B 0,C 180,E1 15100.072,E2 15100.072} C_VEL
LIN {X 0,Y 455.15,Z 874.437,A -85,B 0,C 180,E1 15099.572,E2 15099.572} C_VEL
LIN {X 0,Y 449.899,Z 895.399,A -85,B 0,C 180,E1 15098.972,E2 15098.972} C_VEL
LIN {X 0,Y 443.042,Z 918.881,A -85,B 0,C 180,E1 15098.155,E2 15098.155} C_VEL
LIN {X 0,Y 433.937,Z 945.388,A -85,B 0,C 180,E1 15097,E2 15097} C_VEL
LIN {X 0,Y 425.997,Z 965.774,A -85,B 0,C 180,E1 15095.926,E2 15095.926} C_VEL
LIN {X 0,Y 417.874,Z 984.781,A -85,B 0,C 180,E1 15094.749,E2 15094.749} C_VEL
LIN {X 0,Y 408.844,Z 1004.114,A -85,B 0,C 180,E1 15093.362,E2 15093.362} C_VEL
LIN {X 0,Y 397.358,Z 1026.858,A -85,B 0,C 180,E1 15091.423,E2 15091.423} C_VEL
LIN {X 0,Y 385.671,Z 1047.828,A -85,B 0,C 180,E1 15089.251,E2 15089.251} C_VEL
LIN {X 0,Y 375.822,Z 1064.543,A -85,B 0,C 180,E1 15087.214,E2 15087.214} C_VEL
LIN {X 0,Y 365.879,Z 1080.645,A -85,B 0,C 180,E1 15084.931,E2 15084.931} C_VEL
LIN {X 0,Y 354.336,Z 1098.651,A -85,B 0,C 180,E1 15081.931,E2 15081.931} C_VEL
LIN {X 0,Y 343.012,Z 1115.471,A -85,B 0,C 180,E1 15078.516,E2 15078.516} C_VEL
LIN {X 0,Y 334.189,Z 1128.459,A -85,B 0,C 180,E1 15075.403,E2 15075.403} C_VEL
LIN {X 0,Y 326.255,Z 1140.181,A -85,B 0,C 180,E1 15072.126,E2 15072.126} C_VEL
LIN {X 0,Y 317.575,Z 1153.349,A -85,B 0,C 180,E1 15067.788,E2 15067.788} C_VEL
LIN {X 0,Y 310.124,Z 1165.044,A -85,B 0,C 180,E1 15063.015,E2 15063.015} C_VEL
LIN {X 0,Y 305.317,Z 1173.293,A -85,B 0,C 180,E1 15058.991,E2 15058.991} C_VEL
LIN {X 0,Y 301.646,Z 1180.351,A -85,B 0,C 180,E1 15054.895,E2 15054.895} C_VEL
LIN {X 0,Y 298.885,Z 1186.623,A -85,B 0,C 180,E1 15050.493,E2 15050.493} C_VEL
LIN {X 0,Y 296.91,Z 1192.652,A -85,B 0,C 180,E1 15045.029,E2 15045.029} C_VEL
LIN {X 0,Y 296.184,Z 1196.189,A -85,B 0,C 180,E1 15040.503,E2 15040.503} C_VEL
LIN {X 0,Y 295.998,Z 1198.271,A -85,B 0,C 180,E1 15036.595,E2 15036.595} C_VEL
LIN {X 0,Y 295.986,Z 1199.407,A -85,B 0,C 180,E1 15032.711,E2 15032.711} C_VEL
LIN {X 0,Y 295.992,Z 1199.596,A -85,B 0,C 180,E1 15028.839,E2 15028.839} C_VEL
LIN {X 0,Y 295.981,Z 1198.837,A -85,B 0,C 180,E1 15024.961,E2 15024.961} C_VEL
LIN {X 0,Y 296.073,Z 1197.13,A -85,B 0,C 180,E1 15021.063,E2 15021.063} C_VEL
LIN {X 0,Y 296.496,Z 1194.306,A -85,B 0,C 180,E1 15016.942,E2 15016.942} C_VEL
LIN {X 0,Y 297.526,Z 1190.423,A -85,B 0,C 180,E1 15012.799,E2 15012.799} C_VEL
LIN {X 0,Y 299.347,Z 1185.46,A -85,B 0,C 180,E1 15008.649,E2 15008.649} C_VEL
LIN {X 0,Y 302.095,Z 1179.388,A -85,B 0,C 180,E1 15004.516,E2 15004.516} C_VEL
LIN {X 0,Y 306.139,Z 1171.807,A -85,B 0,C 180,E1 15000.236,E2 15000.236} C_VEL
LIN {X 0,Y 313.094,Z 1160.21,A -85,B 0,C 180,E1 14994.913,E2 14994.913} C_VEL
LIN {X 0,Y 320.04,Z 1149.421,A -85,B 0,C 180,E1 14990.87,E2 14990.87} C_VEL
LIN {X 0,Y 327.258,Z 1138.616,A -85,B 0,C 180,E1 14987.421,E2 14987.421} C_VEL
LIN {X 0,Y 335.514,Z 1126.453,A -85,B 0,C 180,E1 14984.094,E2 14984.094} C_VEL
LIN {X 0,Y 346.496,Z 1110.324,A -85,B 0,C 180,E1 14980.377,E2 14980.377} C_VEL
LIN {X 0,Y 357.057,Z 1094.266,A -85,B 0,C 180,E1 14977.319,E2 14977.319} C_VEL
LIN {X 0,Y 366.751,Z 1079.123,A -85,B 0,C 180,E1 14974.855,E2 14974.855} C_VEL
LIN {X 0,Y 376.434,Z 1063.388,A -85,B 0,C 180,E1 14972.649,E2 14972.649} C_VEL
LIN {X 0,Y 386.967,Z 1045.432,A -85,B 0,C 180,E1 14970.492,E2 14970.492} C_VEL
LIN {X 0,Y 399.734,Z 1021.996,A -85,B 0,C 180,E1 14968.152,E2 14968.152} C_VEL
LIN {X 0,Y 409.5,Z 1002.484,A -85,B 0,C 180,E1 14966.525,E2 14966.525} C_VEL
LIN {X 0,Y 418.264,Z 983.616,A -85,B 0,C 180,E1 14965.184,E2 14965.184} C_VEL
LIN {X 0,Y 426.729,Z 963.69,A -85,B 0,C 180,E1 14963.965,E2 14963.965} C_VEL
LIN {X 0,Y 436.605,Z 937.719,A -85,B 0,C 180,E1 14962.647,E2 14962.647} C_VEL
LIN {X 0,Y 443.967,Z 915.343,A -85,B 0,C 180,E1 14961.722,E2 14961.722} C_VEL
LIN {X 0,Y 450.096,Z 894.104,A -85,B 0,C 180,E1 14960.995,E2 14960.995} C_VEL
LIN {X 0,Y 455.334,Z 872.989,A -85,B 0,C 180,E1 14960.398,E2 14960.398} C_VEL
LIN {X 0,Y 460.127,Z 849.865,A -85,B 0,C 180,E1 14959.876,E2 14959.876} C_VEL
LIN {X 0,Y 464.68,Z 819.544,A -85,B 0,C 180,E1 14959.319,E2 14959.319} C_VEL
LIN {X 0,Y 470.497,Z 756.067,A -85,B 0,C 180,E1 14958.336,E2 14958.336} C_VEL
LIN {X 0,Y 487.318,Z 567.951,A -85,B 0,C 180,E1 14955.486,E2 14955.486} C_VEL
LIN {X 0,Y 482.685,Z 558.565,A -85,B 0,C 180,E1 14952.806,E2 14952.806} C_VEL
LIN {X 0,Y 479.244,Z 552.925,A -85,B 0,C 180,E1 14950.458,E2 14950.458} C_VEL
LIN {X 0,Y 477.381,Z 549.776,A -85,B 0,C 180,E1 14948.917,E2 14948.917} C_VEL
LIN {X 0,Y 474.9,Z 545.451,A -85,B 0,C 180,E1 14946.286,E2 14946.286} C_VEL
LIN {X 0,Y 472.812,Z 541.896,A -85,B 0,C 180,E1 14942.545,E2 14942.545} C_VEL
LIN {X 0,Y 472.574,Z 540.496,A -85,B 0,C 180,E1 14941.212,E2 14941.212} C_VEL
LIN {X 0,Y 472.623,Z 540.751,A -85,B 0,C 180,E1 14937.939,E2 14937.939} C_VEL
LIN {X 0,Y 474.584,Z 545.168,A -85,B 0,C 180,E1 14933.589,E2 14933.589} C_VEL
LIN {X 0,Y 475.262,Z 546.189,A -85,B 0,C 180,E1 14932.748,E2 14932.748} C_VEL
LIN {X 0,Y 478.11,Z 551.015,A -85,B 0,C 180,E1 14929.943,E2 14929.943} C_VEL
LIN {X 0,Y 481.188,Z 556.224,A -85,B 0,C 180,E1 14927.641,E2 14927.641} C_VEL
LIN {X 0,Y 484.814,Z 562.229,A -85,B 0,C 180,E1 14925.427,E2 14925.427} C_VEL
LIN {X 0,Y 487.213,Z 566.675,A -85,B 0,C 180,E1 14924.12,E2 14924.12} C_VEL
LIN {X 0,Y 467.07,Z 792.018,A -85,B 0,C 180,E1 14920.713,E2 14920.713} C_VEL
LIN {X 0,Y 463.668,Z 821.386,A -85,B 0,C 180,E1 14920.228,E2 14920.228} C_VEL
LIN {X 0,Y 459.943,Z 843.718,A -85,B 0,C 180,E1 14919.776,E2 14919.776} C_VEL
LIN {X 0,Y 455.528,Z 864.973,A -85,B 0,C 180,E1 14919.235,E2 14919.235} C_VEL
LIN {X 0,Y 450.094,Z 886.806,A -85,B 0,C 180,E1 14918.557,E2 14918.557} C_VEL
LIN {X 0,Y 442.049,Z 913.92,A -85,B 0,C 180,E1 14917.514,E2 14917.514} C_VEL
LIN {X 0,Y 434.493,Z 935.573,A -85,B 0,C 180,E1 14916.495,E2 14916.495} C_VEL
LIN {X 0,Y 426.714,Z 955.522,A -85,B 0,C 180,E1 14915.387,E2 14915.387} C_VEL
LIN {X 0,Y 418.356,Z 974.901,A -85,B 0,C 180,E1 14914.135,E2 14914.135} C_VEL
LIN {X 0,Y 407.775,Z 997.346,A -85,B 0,C 180,E1 14912.423,E2 14912.423} C_VEL
LIN {X 0,Y 396.288,Z 1019.111,A -85,B 0,C 180,E1 14910.414,E2 14910.414} C_VEL
LIN {X 0,Y 386.685,Z 1036.083,A -85,B 0,C 180,E1 14908.571,E2 14908.571} C_VEL
LIN {X 0,Y 377.264,Z 1051.771,A -85,B 0,C 180,E1 14906.599,E2 14906.599} C_VEL
LIN {X 0,Y 367.106,Z 1067.83,A -85,B 0,C 180,E1 14904.256,E2 14904.256} C_VEL
LIN {X 0,Y 354.329,Z 1087.015,A -85,B 0,C 180,E1 14900.896,E2 14900.896} C_VEL
LIN {X 0,Y 344.64,Z 1100.939,A -85,B 0,C 180,E1 14897.962,E2 14897.962} C_VEL
LIN {X 0,Y 336.254,Z 1112.782,A -85,B 0,C 180,E1 14895.048,E2 14895.048} C_VEL
LIN {X 0,Y 328.255,Z 1123.981,A -85,B 0,C 180,E1 14891.841,E2 14891.841} C_VEL
LIN {X 0,Y 319.568,Z 1136.322,A -85,B 0,C 180,E1 14887.664,E2 14887.664} C_VEL
LIN {X 0,Y 311.918,Z 1147.404,A -85,B 0,C 180,E1 14883.02,E2 14883.02} C_VEL
LIN {X 0,Y 306.841,Z 1155.266,A -85,B 0,C 180,E1 14879.047,E2 14879.047} C_VEL
LIN {X 0,Y 302.891,Z 1161.969,A -85,B 0,C 180,E1 14874.995,E2 14874.995} C_VEL
LIN {X 0,Y 299.957,Z 1167.565,A -85,B 0,C 180,E1 14870.896,E2 14870.896} C_VEL
LIN {X 0,Y 297.844,Z 1172.496,A -85,B 0,C 180,E1 14866.379,E2 14866.379} C_VEL
LIN {X 0,Y 296.538,Z 1176.703,A -85,B 0,C 180,E1 14861.081,E2 14861.081} C_VEL
LIN {X 0,Y 296.115,Z 1178.945,A -85,B 0,C 180,E1 14856.592,E2 14856.592} C_VEL
LIN {X 0,Y 296.001,Z 1179.992,A -85,B 0,C 180,E1 14852.711,E2 14852.711} C_VEL
LIN {X 0,Y 295.994,Z 1180.176,A -85,B 0,C 180,E1 14848.839,E2 14848.839} C_VEL
LIN {X 0,Y 296.042,Z 1179.501,A -85,B 0,C 180,E1 14844.962,E2 14844.962} C_VEL
LIN {X 0,Y 296.292,Z 1177.849,A -85,B 0,C 180,E1 14840.874,E2 14840.874} C_VEL
LIN {X 0,Y 296.928,Z 1175.182,A -85,B 0,C 180,E1 14836.705,E2 14836.705} C_VEL
LIN {X 0,Y 298.185,Z 1171.606,A -85,B 0,C 180,E1 14832.637,E2 14832.637} C_VEL
LIN {X 0,Y 300.269,Z 1166.957,A -85,B 0,C 180,E1 14828.513,E2 14828.513} C_VEL
LIN {X 0,Y 303.487,Z 1160.949,A -85,B 0,C 180,E1 14824.222,E2 14824.222} C_VEL
LIN {X 0,Y 308.797,Z 1152.337,A -85,B 0,C 180,E1 14819.23,E2 14819.23} C_VEL
LIN {X 0,Y 315.567,Z 1142.032,A -85,B 0,C 180,E1 14814.52,E2 14814.52} C_VEL
LIN {X 0,Y 322.456,Z 1132.186,A -85,B 0,C 180,E1 14810.761,E2 14810.761} C_VEL
LIN {X 0,Y 330.534,Z 1120.884,A -85,B 0,C 180,E1 14807.108,E2 14807.108} C_VEL
LIN {X 0,Y 342.064,Z 1104.711,A -85,B 0,C 180,E1 14802.805,E2 14802.805} C_VEL
LIN {X 0,Y 351.513,Z 1091.165,A -85,B 0,C 180,E1 14799.826,E2 14799.826} C_VEL
LIN {X 0,Y 360.654,Z 1077.697,A -85,B 0,C 180,E1 14797.282,E2 14797.282} C_VEL
LIN {X 0,Y 371.021,Z 1061.868,A -85,B 0,C 180,E1 14794.721,E2 14794.721} C_VEL
LIN {X 0,Y 383.942,Z 1040.972,A -85,B 0,C 180,E1 14791.901,E2 14791.901} C_VEL
LIN {X 0,Y 394.316,Z 1022.871,A -85,B 0,C 180,E1 14789.865,E2 14789.865} C_VEL
LIN {X 0,Y 397.09,Z 1017.894,A -85,B 0,C 180,E1 14789.36,E2 14789.36} C_VEL
LIN {X 0,Y 399.706,Z 1012.316,A -85,B 0,C 180,E1 14788.682,E2 14788.682} C_VEL
LIN {X 0,Y 404.386,Z 997.907,A -85,B 0,C 180,E1 14786.571,E2 14786.571} C_VEL
LIN {X 0,Y 406.597,Z 992.718,A -85,B 0,C 180,E1 14786.061,E2 14786.061} C_VEL
LIN {X 0,Y 415.427,Z 974.267,A -85,B 0,C 180,E1 14784.691,E2 14784.691} C_VEL
LIN {X 0,Y 423.545,Z 955.786,A -85,B 0,C 180,E1 14783.514,E2 14783.514} C_VEL
LIN {X 0,Y 431.273,Z 936.374,A -85,B 0,C 180,E1 14782.446,E2 14782.446} C_VEL
LIN {X 0,Y 440.024,Z 911.765,A -85,B 0,C 180,E1 14781.31,E2 14781.31} C_VEL
LIN {X 0,Y 447.62,Z 886.169,A -85,B 0,C 180,E1 14780.357,E2 14780.357} C_VEL
LIN {X 0,Y 453.049,Z 864.62,A -85,B 0,C 180,E1 14779.7,E2 14779.7} C_VEL
LIN {X 0,Y 457.524,Z 843.328,A -85,B 0,C 180,E1 14779.169,E2 14779.169} C_VEL
LIN {X 0,Y 461.464,Z 819.869,A -85,B 0,C 180,E1 14778.706,E2 14778.706} C_VEL
LIN {X 0,Y 465.39,Z 784.063,A -85,B 0,C 180,E1 14778.133,E2 14778.133} C_VEL
LIN {X 0,Y 484.757,Z 572.322,A -85,B 0,C 180,E1 14774.95,E2 14774.95} C_VEL
LIN {X 0,Y 480.865,Z 565.457,A -85,B 0,C 180,E1 14772.611,E2 14772.611} C_VEL
LIN {X 0,Y 478.145,Z 560.884,A -85,B 0,C 180,E1 14770.665,E2 14770.665} C_VEL
LIN {X 0,Y 476.283,Z 557.566,A -85,B 0,C 180,E1 14769.059,E2 14769.059} C_VEL
LIN {X 0,Y 473.813,Z 553.281,A -85,B 0,C 180,E1 14766.3,E2 14766.3} C_VEL
LIN {X 0,Y 471.861,Z 549.151,A -85,B 0,C 180,E1 14761.943,E2 14761.943} C_VEL
LIN {X 0,Y 471.783,Z 548.48,A -85,B 0,C 180,E1 14761.093,E2 14761.093} C_VEL
LIN {X 0,Y 471.838,Z 548.763,A -85,B 0,C 180,E1 14758.786,E2 14758.786} C_VEL
LIN {X 0,Y 473.404,Z 552.838,A -85,B 0,C 180,E1 14754.668,E2 14754.668} C_VEL
LIN {X 0,Y 474.325,Z 554.057,A -85,B 0,C 180,E1 14753.464,E2 14753.464} C_VEL
LIN {X 0,Y 477.208,Z 559.132,A -85,B 0,C 180,E1 14750.533,E2 14750.533} C_VEL
LIN {X 0,Y 479.813,Z 563.657,A -85,B 0,C 180,E1 14748.521,E2 14748.521} C_VEL
LIN {X 0,Y 482.167,Z 567.866,A -85,B 0,C 180,E1 14746.967,E2 14746.967} C_VEL
LIN {X 0,Y 484.851,Z 573.763,A -85,B 0,C 180,E1 14745.343,E2 14745.343} C_VEL
LIN {X 0,Y 464.645,Z 795.558,A -85,B 0,C 180,E1 14742.005,E2 14742.005} C_VEL
LIN {X 0,Y 460.778,Z 830.378,A -85,B 0,C 180,E1 14741.439,E2 14741.439} C_VEL
LIN {X 0,Y 456.806,Z 853.68,A -85,B 0,C 180,E1 14740.997,E2 14740.997} C_VEL
LIN {X 0,Y 452.145,Z 875.258,A -85,B 0,C 180,E1 14740.503,E2 14740.503} C_VEL
LIN {X 0,Y 446.256,Z 898.114,A -85,B 0,C 180,E1 14739.849,E2 14739.849} C_VEL
LIN {X 0,Y 437.568,Z 926.187,A -85,B 0,C 180,E1 14738.835,E2 14738.835} C_VEL
LIN {X 0,Y 430.035,Z 947.149,A -85,B 0,C 180,E1 14737.901,E2 14737.901} C_VEL
LIN {X 0,Y 422.34,Z 966.417,A -85,B 0,C 180,E1 14736.888,E2 14736.888} C_VEL
LIN {X 0,Y 414.059,Z 985.334,A -85,B 0,C 180,E1 14735.724,E2 14735.724} C_VEL
LIN {X 0,Y 404.485,Z 1005.33,A -85,B 0,C 180,E1 14734.292,E2 14734.292} C_VEL
LIN {X 0,Y 391.351,Z 1030.291,A -85,B 0,C 180,E1 14732.124,E2 14732.124} C_VEL
LIN {X 0,Y 380.808,Z 1048.68,A -85,B 0,C 180,E1 14730.2,E2 14730.2} C_VEL
LIN {X 0,Y 370.724,Z 1065.298,A -85,B 0,C 180,E1 14728.164,E2 14728.164} C_VEL
LIN {X 0,Y 359.619,Z 1082.719,A -85,B 0,C 180,E1 14725.665,E2 14725.665} C_VEL
LIN {X 0,Y 346.977,Z 1101.519,A -85,B 0,C 180,E1 14722.415,E2 14722.415} C_VEL
LIN {X 0,Y 336.97,Z 1115.909,A -85,B 0,C 180,E1 14719.429,E2 14719.429} C_VEL
LIN {X 0,Y 328.305,Z 1128.183,A -85,B 0,C 180,E1 14716.455,E2 14716.455} C_VEL
LIN {X 0,Y 319.53,Z 1140.623,A -85,B 0,C 180,E1 14712.925,E2 14712.925} C_VEL
LIN {X 0,Y 310.051,Z 1154.326,A -85,B 0,C 180,E1 14708.255,E2 14708.255} C_VEL
LIN {X 0,Y 303.095,Z 1164.769,A -85,B 0,C 180,E1 14703.883,E2 14703.883} C_VEL
LIN {X 0,Y 298.003,Z 1173.019,A -85,B 0,C 180,E1 14699.773,E2 14699.773} C_VEL
LIN {X 0,Y 294.092,Z 1180.078,A -85,B 0,C 180,E1 14695.58,E2 14695.58} C_VEL
LIN {X 0,Y 291.187,Z 1186.26,A -85,B 0,C 180,E1 14691.133,E2 14691.133} C_VEL
LIN {X 0,Y 289.06,Z 1192.217,A -85,B 0,C 180,E1 14685.652,E2 14685.652} C_VEL
LIN {X 0,Y 288.208,Z 1195.922,A -85,B 0,C 180,E1 14680.797,E2 14680.797} C_VEL
LIN {X 0,Y 288.003,Z 1198.007,A -85,B 0,C 180,E1 14676.779,E2 14676.779} C_VEL
LIN {X 0,Y 287.99,Z 1199.145,A -85,B 0,C 180,E1 14672.786,E2 14672.786} C_VEL
LIN {X 0,Y 287.996,Z 1199.334,A -85,B 0,C 180,E1 14668.806,E2 14668.806} C_VEL
LIN {X 0,Y 287.985,Z 1198.574,A -85,B 0,C 180,E1 14664.821,E2 14664.821} C_VEL
LIN {X 0,Y 288.089,Z 1196.865,A -85,B 0,C 180,E1 14660.813,E2 14660.813} C_VEL
LIN {X 0,Y 288.554,Z 1194.038,A -85,B 0,C 180,E1 14656.576,E2 14656.576} C_VEL
LIN {X 0,Y 289.599,Z 1190.367,A -85,B 0,C 180,E1 14652.52,E2 14652.52} C_VEL
LIN {X 0,Y 291.523,Z 1185.451,A -85,B 0,C 180,E1 14648.259,E2 14648.259} C_VEL
LIN {X 0,Y 294.415,Z 1179.426,A -85,B 0,C 180,E1 14644.018,E2 14644.018} C_VEL
LIN {X 0,Y 298.461,Z 1172.215,A -85,B 0,C 180,E1 14639.808,E2 14639.808} C_VEL
LIN {X 0,Y 305.048,Z 1161.808,A -85,B 0,C 180,E1 14634.769,E2 14634.769} C_VEL
LIN {X 0,Y 313.162,Z 1149.669,A -85,B 0,C 180,E1 14630.078,E2 14630.078} C_VEL
LIN {X 0,Y 320.574,Z 1139.052,A -85,B 0,C 180,E1 14626.614,E2 14626.614} C_VEL
LIN {X 0,Y 329.224,Z 1126.822,A -85,B 0,C 180,E1 14623.207,E2 14623.207} C_VEL
LIN {X 0,Y 340.573,Z 1110.824,A -85,B 0,C 180,E1 14619.456,E2 14619.456} C_VEL
LIN {X 0,Y 352.124,Z 1093.831,A -85,B 0,C 180,E1 14616.202,E2 14616.202} C_VEL
LIN {X 0,Y 362.022,Z 1078.845,A -85,B 0,C 180,E1 14613.765,E2 14613.765} C_VEL
LIN {X 0,Y 371.586,Z 1063.76,A -85,B 0,C 180,E1 14611.65,E2 14611.65} C_VEL
LIN {X 0,Y 381.798,Z 1046.84,A -85,B 0,C 180,E1 14609.606,E2 14609.606} C_VEL
LIN {X 0,Y 394.14,Z 1025.088,A -85,B 0,C 180,E1 14607.392,E2 14607.392} C_VEL
LIN {X 0,Y 405.239,Z 1003.518,A -85,B 0,C 180,E1 14605.582,E2 14605.582} C_VEL
LIN {X 0,Y 414.413,Z 984.255,A -85,B 0,C 180,E1 14604.216,E2 14604.216} C_VEL
LIN {X 0,Y 422.704,Z 965.229,A -85,B 0,C 180,E1 14603.055,E2 14603.055} C_VEL
LIN {X 0,Y 431.535,Z 942.906,A -85,B 0,C 180,E1 14601.904,E2 14601.904} C_VEL
LIN {X 0,Y 440.63,Z 916.36,A -85,B 0,C 180,E1 14600.79,E2 14600.79} C_VEL
LIN {X 0,Y 447.038,Z 894.646,A -85,B 0,C 180,E1 14600.052,E2 14600.052} C_VEL
LIN {X 0,Y 452.418,Z 873.423,A -85,B 0,C 180,E1 14599.458,E2 14599.458} C_VEL
LIN {X 0,Y 457.143,Z 851.157,A -85,B 0,C 180,E1 14598.959,E2 14598.959} C_VEL
LIN {X 0,Y 461.68,Z 822.886,A -85,B 0,C 180,E1 14598.435,E2 14598.435} C_VEL
LIN {X 0,Y 466.212,Z 776.089,A -85,B 0,C 180,E1 14597.708,E2 14597.708} C_VEL
LIN {X 0,Y 484.689,Z 573.384,A -85,B 0,C 180,E1 14594.652,E2 14594.652} C_VEL
LIN {X 0,Y 480.941,Z 565.702,A -85,B 0,C 180,E1 14592.365,E2 14592.365} C_VEL
LIN {X 0,Y 477.947,Z 560.612,A -85,B 0,C 180,E1 14590.243,E2 14590.243} C_VEL
LIN {X 0,Y 476.13,Z 557.49,A -85,B 0,C 180,E1 14588.697,E2 14588.697} C_VEL
LIN {X 0,Y 473.726,Z 553.238,A -85,B 0,C 180,E1 14586.058,E2 14586.058} C_VEL
LIN {X 0,Y 471.77,Z 549.625,A -85,B 0,C 180,E1 14582.308,E2 14582.308} C_VEL
LIN {X 0,Y 471.575,Z 548.439,A -85,B 0,C 180,E1 14581.093,E2 14581.093} C_VEL
LIN {X 0,Y 471.626,Z 548.634,A -85,B 0,C 180,E1 14578.056,E2 14578.056} C_VEL
LIN {X 0,Y 473.516,Z 553.051,A -85,B 0,C 180,E1 14573.696,E2 14573.696} C_VEL
LIN {X 0,Y 474.176,Z 554.108,A -85,B 0,C 180,E1 14572.853,E2 14572.853} C_VEL
LIN {X 0,Y 476.843,Z 558.706,A -85,B 0,C 180,E1 14570.16,E2 14570.16} C_VEL
LIN {X 0,Y 479.848,Z 563.921,A -85,B 0,C 180,E1 14567.851,E2 14567.851} C_VEL
LIN {X 0,Y 483.304,Z 569.775,A -85,B 0,C 180,E1 14565.686,E2 14565.686} C_VEL
LIN {X 0,Y 484.572,Z 572.411,A -85,B 0,C 180,E1 14564.949,E2 14564.949} C_VEL
LIN {X 0,Y 464.028,Z 797.098,A -85,B 0,C 180,E1 14561.572,E2 14561.572} C_VEL
LIN {X 0,Y 460.811,Z 823.03,A -85,B 0,C 180,E1 14561.14,E2 14561.14} C_VEL
LIN {X 0,Y 457.064,Z 844.88,A -85,B 0,C 180,E1 14560.699,E2 14560.699} C_VEL
LIN {X 0,Y 452.449,Z 866.543,A -85,B 0,C 180,E1 14560.149,E2 14560.149} C_VEL
LIN {X 0,Y 445.853,Z 892.225,A -85,B 0,C 180,E1 14559.343,E2 14559.343} C_VEL
LIN {X 0,Y 437.86,Z 917.564,A -85,B 0,C 180,E1 14558.339,E2 14558.339} C_VEL
LIN {X 0,Y 430.566,Z 937.841,A -85,B 0,C 180,E1 14557.379,E2 14557.379} C_VEL
LIN {X 0,Y 422.652,Z 957.58,A -85,B 0,C 180,E1 14556.279,E2 14556.279} C_VEL
LIN {X 0,Y 413.048,Z 979.193,A -85,B 0,C 180,E1 14554.868,E2 14554.868} C_VEL
LIN {X 0,Y 401.208,Z 1002.952,A -85,B 0,C 180,E1 14552.99,E2 14552.99} C_VEL
LIN {X 0,Y 391.4,Z 1020.967,A -85,B 0,C 180,E1 14551.297,E2 14551.297} C_VEL
LIN {X 0,Y 381.799,Z 1037.454,A -85,B 0,C 180,E1 14549.495,E2 14549.495} C_VEL
LIN {X 0,Y 371.912,Z 1053.429,A -85,B 0,C 180,E1 14547.472,E2 14547.472} C_VEL
LIN {X 0,Y 359.669,Z 1072.184,A -85,B 0,C 180,E1 14544.673,E2 14544.673} C_VEL
LIN {X 0,Y 347.996,Z 1088.878,A -85,B 0,C 180,E1 14541.638,E2 14541.638} C_VEL
LIN {X 0,Y 338.423,Z 1102.165,A -85,B 0,C 180,E1 14538.786,E2 14538.786} C_VEL
LIN {X 0,Y 329.493,Z 1114.307,A -85,B 0,C 180,E1 14535.736,E2 14535.736} C_VEL
LIN {X 0,Y 319.646,Z 1127.625,A -85,B 0,C 180,E1 14531.779,E2 14531.779} C_VEL
LIN {X 0,Y 310.523,Z 1139.931,A -85,B 0,C 180,E1 14527.253,E2 14527.253} C_VEL
LIN {X 0,Y 304.128,Z 1148.861,A -85,B 0,C 180,E1 14523.301,E2 14523.301} C_VEL
LIN {X 0,Y 298.934,Z 1156.569,A -85,B 0,C 180,E1 14519.231,E2 14519.231} C_VEL
LIN {X 0,Y 294.573,Z 1163.71,A -85,B 0,C 180,E1 14514.676,E2 14514.676} C_VEL
LIN {X 0,Y 290.958,Z 1170.578,A -85,B 0,C 180,E1 14509.054,E2 14509.054} C_VEL
LIN {X 0,Y 289.275,Z 1174.677,A -85,B 0,C 180,E1 14504.571,E2 14504.571} C_VEL
LIN {X 0,Y 288.444,Z 1177.511,A -85,B 0,C 180,E1 14500.384,E2 14500.384} C_VEL
LIN {X 0,Y 288.109,Z 1179.338,A -85,B 0,C 180,E1 14496.376,E2 14496.376} C_VEL
LIN {X 0,Y 288.003,Z 1180.276,A -85,B 0,C 180,E1 14492.587,E2 14492.587} C_VEL
LIN {X 0,Y 287.999,Z 1180.417,A -85,B 0,C 180,E1 14488.607,E2 14488.607} C_VEL
LIN {X 0,Y 288.058,Z 1179.699,A -85,B 0,C 180,E1 14484.623,E2 14484.623} C_VEL
LIN {X 0,Y 288.323,Z 1178.113,A -85,B 0,C 180,E1 14480.62,E2 14480.62} C_VEL
LIN {X 0,Y 289.005,Z 1175.493,A -85,B 0,C 180,E1 14476.393,E2 14476.393} C_VEL
LIN {X 0,Y 290.381,Z 1171.874,A -85,B 0,C 180,E1 14472.155,E2 14472.155} C_VEL
LIN {X 0,Y 292.619,Z 1167.227,A -85,B 0,C 180,E1 14467.922,E2 14467.922} C_VEL
LIN {X 0,Y 296.062,Z 1161.194,A -85,B 0,C 180,E1 14463.507,E2 14463.507} C_VEL
LIN {X 0,Y 301.706,Z 1152.567,A -85,B 0,C 180,E1 14458.401,E2 14458.401} C_VEL
LIN {X 0,Y 308.757,Z 1142.388,A -85,B 0,C 180,E1 14453.657,E2 14453.657} C_VEL
LIN {X 0,Y 315.665,Z 1132.961,A -85,B 0,C 180,E1 14449.985,E2 14449.985} C_VEL
LIN {X 0,Y 323.612,Z 1122.279,A -85,B 0,C 180,E1 14446.449,E2 14446.449} C_VEL
LIN {X 0,Y 334.059,Z 1108.333,A -85,B 0,C 180,E1 14442.567,E2 14442.567} C_VEL
LIN {X 0,Y 345.175,Z 1092.951,A -85,B 0,C 180,E1 14439.076,E2 14439.076} C_VEL
LIN {X 0,Y 355.114,Z 1078.799,A -85,B 0,C 180,E1 14436.365,E2 14436.365} C_VEL
LIN {X 0,Y 365.147,Z 1063.962,A -85,B 0,C 180,E1 14433.934,E2 14433.934} C_VEL
LIN {X 0,Y 376.411,Z 1046.498,A -85,B 0,C 180,E1 14431.497,E2 14431.497} C_VEL
LIN {X 0,Y 388.938,Z 1025.543,A -85,B 0,C 180,E1 14429.068,E2 14429.068} C_VEL
LIN {X 0,Y 399.022,Z 1007.317,A -85,B 0,C 180,E1 14427.295,E2 14427.295} C_VEL
LIN {X 0,Y 406.597,Z 992.718,A -85,B 0,C 180,E1 14426.061,E2 14426.061} C_VEL
LIN {X 0,Y 409.178,Z 986.717,A -85,B 0,C 180,E1 14425.472,E2 14425.472} C_VEL
LIN {X 0,Y 412.405,Z 976.265,A -85,B 0,C 180,E1 14424.135,E2 14424.135} C_VEL
LIN {X 0,Y 414.594,Z 969.552,A -85,B 0,C 180,E1 14423.384,E2 14423.384} C_VEL
LIN {X 0,Y 416.134,Z 965.951,A -85,B 0,C 180,E1 14423.099,E2 14423.099} C_VEL
LIN {X 0,Y 426.189,Z 941.936,A -85,B 0,C 180,E1 14421.716,E2 14421.716} C_VEL
LIN {X 0,Y 433.596,Z 922.134,A -85,B 0,C 180,E1 14420.761,E2 14420.761} C_VEL
LIN {X 0,Y 440.315,Z 901.891,A -85,B 0,C 180,E1 14419.932,E2 14419.932} C_VEL
LIN {X 0,Y 446.306,Z 881.196,A -85,B 0,C 180,E1 14419.217,E2 14419.217} C_VEL
LIN {X 0,Y 452.357,Z 856.553,A -85,B 0,C 180,E1 14418.517,E2 14418.517} C_VEL
LIN {X 0,Y 457.592,Z 828.848,A -85,B 0,C 180,E1 14417.916,E2 14417.916} C_VEL
LIN {X 0,Y 460.769,Z 805.915,A -85,B 0,C 180,E1 14417.524,E2 14417.524} C_VEL
LIN {X 0,Y 480.8,Z 593.064,A -85,B 0,C 180,E1 14414.338,E2 14414.338} C_VEL
LIN {X 0,Y 482.216,Z 577.956,A -85,B 0,C 180,E1 14414.102,E2 14414.102} C_VEL
LIN {X 0,Y 478.911,Z 572.148,A -85,B 0,C 180,E1 14411.99,E2 14411.99} C_VEL
LIN {X 0,Y 476.711,Z 568.33,A -85,B 0,C 180,E1 14410.331,E2 14410.331} C_VEL
LIN {X 0,Y 475.043,Z 565.285,A -85,B 0,C 180,E1 14408.839,E2 14408.839} C_VEL
LIN {X 0,Y 472.746,Z 561.164,A -85,B 0,C 180,E1 14406.192,E2 14406.192} C_VEL
LIN {X 0,Y 470.864,Z 557.032,A -85,B 0,C 180,E1 14401.825,E2 14401.825} C_VEL
LIN {X 0,Y 470.794,Z 556.417,A -85,B 0,C 180,E1 14400.974,E2 14400.974} C_VEL
LIN {X 0,Y 470.847,Z 556.641,A -85,B 0,C 180,E1 14398.905,E2 14398.905} C_VEL
LIN {X 0,Y 472.345,Z 560.721,A -85,B 0,C 180,E1 14394.777,E2 14394.777} C_VEL
LIN {X 0,Y 473.242,Z 561.977,A -85,B 0,C 180,E1 14393.57,E2 14393.57} C_VEL
LIN {X 0,Y 476.01,Z 566.953,A -85,B 0,C 180,E1 14390.692,E2 14390.692} C_VEL
LIN {X 0,Y 478.485,Z 571.353,A -85,B 0,C 180,E1 14388.733,E2 14388.733} C_VEL
LIN {X 0,Y 480.652,Z 575.326,A -85,B 0,C 180,E1 14387.261,E2 14387.261} C_VEL
LIN {X 0,Y 482.333,Z 579.185,A -85,B 0,C 180,E1 14386.185,E2 14386.185} C_VEL
LIN {X 0,Y 461.698,Z 801.072,A -85,B 0,C 180,E1 14382.868,E2 14382.868} C_VEL
LIN {X 0,Y 458.152,Z 830.943,A -85,B 0,C 180,E1 14382.379,E2 14382.379} C_VEL
LIN {X 0,Y 454.201,Z 853.659,A -85,B 0,C 180,E1 14381.953,E2 14381.953} C_VEL
LIN {X 0,Y 449.417,Z 875.42,A -85,B 0,C 180,E1 14381.462,E2 14381.462} C_VEL
LIN {X 0,Y 443.125,Z 899.345,A -85,B 0,C 180,E1 14380.785,E2 14380.785} C_VEL
LIN {X 0,Y 434.608,Z 926.181,A -85,B 0,C 180,E1 14379.825,E2 14379.825} C_VEL
LIN {X 0,Y 426.938,Z 947.127,A -85,B 0,C 180,E1 14378.904,E2 14378.904} C_VEL
LIN {X 0,Y 418.805,Z 967.06,A -85,B 0,C 180,E1 14377.867,E2 14377.867} C_VEL
LIN {X 0,Y 410.366,Z 985.887,A -85,B 0,C 180,E1 14376.716,E2 14376.716} C_VEL
LIN {X 0,Y 399.587,Z 1007.858,A -85,B 0,C 180,E1 14375.141,E2 14375.141} C_VEL
LIN {X 0,Y 386.994,Z 1030.962,A -85,B 0,C 180,E1 14373.118,E2 14373.118} C_VEL
LIN {X 0,Y 376.641,Z 1048.57,A -85,B 0,C 180,E1 14371.281,E2 14371.281} C_VEL
LIN {X 0,Y 366.385,Z 1065.027,A -85,B 0,C 180,E1 14369.275,E2 14369.275} C_VEL
LIN {X 0,Y 355.266,Z 1081.978,A -85,B 0,C 180,E1 14366.854,E2 14366.854} C_VEL
LIN {X 0,Y 341.904,Z 1101.245,A -85,B 0,C 180,E1 14363.533,E2 14363.533} C_VEL
LIN {X 0,Y 331.54,Z 1115.634,A -85,B 0,C 180,E1 14360.538,E2 14360.538} C_VEL
LIN {X 0,Y 322.063,Z 1128.555,A -85,B 0,C 180,E1 14357.373,E2 14357.373} C_VEL
LIN {X 0,Y 312.698,Z 1141.31,A -85,B 0,C 180,E1 14353.682,E2 14353.682} C_VEL
LIN {X 0,Y 302.536,Z 1155.296,A -85,B 0,C 180,E1 14348.74,E2 14348.74} C_VEL
LIN {X 0,Y 295.848,Z 1164.909,A -85,B 0,C 180,E1 14344.595,E2 14344.595} C_VEL
LIN {X 0,Y 290.523,Z 1173.108,A -85,B 0,C 180,E1 14340.392,E2 14340.392} C_VEL
LIN {X 0,Y 286.25,Z 1180.431,A -85,B 0,C 180,E1 14335.888,E2 14335.888} C_VEL
LIN {X 0,Y 282.711,Z 1187.749,A -85,B 0,C 180,E1 14330.279,E2 14330.279} C_VEL
LIN {X 0,Y 280.95,Z 1192.616,A -85,B 0,C 180,E1 14325.269,E2 14325.269} C_VEL
LIN {X 0,Y 280.216,Z 1195.776,A -85,B 0,C 180,E1 14320.901,E2 14320.901} C_VEL
LIN {X 0,Y 280.006,Z 1197.815,A -85,B 0,C 180,E1 14316.767,E2 14316.767} C_VEL
LIN {X 0,Y 279.994,Z 1198.882,A -85,B 0,C 180,E1 14312.866,E2 14312.866} C_VEL
LIN {X 0,Y 280,Z 1199.071,A -85,B 0,C 180,E1 14308.772,E2 14308.772} C_VEL
LIN {X 0,Y 279.989,Z 1198.31,A -85,B 0,C 180,E1 14304.673,E2 14304.673} C_VEL
LIN {X 0,Y 280.104,Z 1196.599,A -85,B 0,C 180,E1 14300.549,E2 14300.549} C_VEL
LIN {X 0,Y 280.62,Z 1193.769,A -85,B 0,C 180,E1 14296.189,E2 14296.189} C_VEL
LIN {X 0,Y 281.755,Z 1190.083,A -85,B 0,C 180,E1 14292.005,E2 14292.005} C_VEL
LIN {X 0,Y 283.83,Z 1185.178,A -85,B 0,C 180,E1 14287.638,E2 14287.638} C_VEL
LIN {X 0,Y 286.937,Z 1179.151,A -85,B 0,C 180,E1 14283.288,E2 14283.288} C_VEL
LIN {X 0,Y 291.208,Z 1171.981,A -85,B 0,C 180,E1 14279.001,E2 14279.001} C_VEL
LIN {X 0,Y 298.206,Z 1161.53,A -85,B 0,C 180,E1 14273.835,E2 14273.835} C_VEL
LIN {X 0,Y 306.447,Z 1149.773,A -85,B 0,C 180,E1 14269.199,E2 14269.199} C_VEL
LIN {X 0,Y 314.378,Z 1138.911,A -85,B 0,C 180,E1 14265.598,E2 14265.598} C_VEL
LIN {X 0,Y 323.016,Z 1127.19,A -85,B 0,C 180,E1 14262.286,E2 14262.286} C_VEL
LIN {X 0,Y 333.655,Z 1112.696,A -85,B 0,C 180,E1 14258.818,E2 14258.818} C_VEL
LIN {X 0,Y 346.605,Z 1094.449,A -85,B 0,C 180,E1 14255.237,E2 14255.237} C_VEL
LIN {X 0,Y 357.177,Z 1078.942,A -85,B 0,C 180,E1 14252.703,E2 14252.703} C_VEL
LIN {X 0,Y 367.028,Z 1063.86,A -85,B 0,C 180,E1 14250.588,E2 14250.588} C_VEL
LIN {X 0,Y 377.356,Z 1047.214,A -85,B 0,C 180,E1 14248.581,E2 14248.581} C_VEL
LIN {X 0,Y 390.04,Z 1025.486,A -85,B 0,C 180,E1 14246.372,E2 14246.372} C_VEL
LIN {X 0,Y 401.695,Z 1003.341,A -85,B 0,C 180,E1 14244.527,E2 14244.527} C_VEL
LIN {X 0,Y 410.679,Z 984.903,A -85,B 0,C 180,E1 14243.23,E2 14243.23} C_VEL
LIN {X 0,Y 419.175,Z 965.861,A -85,B 0,C 180,E1 14242.076,E2 14242.076} C_VEL
LIN {X 0,Y 427.412,Z 945.547,A -85,B 0,C 180,E1 14241.03,E2 14241.03} C_VEL
LIN {X 0,Y 436.607,Z 919.961,A -85,B 0,C 180,E1 14239.937,E2 14239.937} C_VEL
LIN {X 0,Y 444.123,Z 895.115,A -85,B 0,C 180,E1 14239.094,E2 14239.094} C_VEL
LIN {X 0,Y 449.667,Z 873.677,A -85,B 0,C 180,E1 14238.502,E2 14238.502} C_VEL
LIN {X 0,Y 454.408,Z 851.795,A -85,B 0,C 180,E1 14238.017,E2 14238.017} C_VEL
LIN {X 0,Y 459.006,Z 824.288,A -85,B 0,C 180,E1 14237.509,E2 14237.509} C_VEL
LIN {X 0,Y 463.465,Z 779.742,A -85,B 0,C 180,E1 14236.819,E2 14236.819} C_VEL
LIN {X 0,Y 482.17,Z 578.844,A -85,B 0,C 180,E1 14233.814,E2 14233.814} C_VEL
LIN {X 0,Y 479.405,Z 573.111,A -85,B 0,C 180,E1 14232.039,E2 14232.039} C_VEL
LIN {X 0,Y 476.583,Z 568.177,A -85,B 0,C 180,E1 14229.967,E2 14229.967} C_VEL
LIN {X 0,Y 474.886,Z 565.203,A -85,B 0,C 180,E1 14228.476,E2 14228.476} C_VEL
LIN {X 0,Y 472.655,Z 561.119,A -85,B 0,C 180,E1 14225.95,E2 14225.95} C_VEL
LIN {X 0,Y 470.759,Z 557.505,A -85,B 0,C 180,E1 14222.191,E2 14222.191} C_VEL
LIN {X 0,Y 470.6,Z 556.38,A -85,B 0,C 180,E1 14221.096,E2 14221.096} C_VEL
LIN {X 0,Y 470.63,Z 556.517,A -85,B 0,C 180,E1 14218.174,E2 14218.174} C_VEL
LIN {X 0,Y 472.543,Z 561.024,A -85,B 0,C 180,E1 14213.683,E2 14213.683} C_VEL
LIN {X 0,Y 473.578,Z 563.1,A -85,B 0,C 180,E1 14212.356,E2 14212.356} C_VEL
LIN {X 0,Y 475.583,Z 566.396,A -85,B 0,C 180,E1 14210.378,E2 14210.378} C_VEL
LIN {X 0,Y 478.516,Z 571.617,A -85,B 0,C 180,E1 14208.061,E2 14208.061} C_VEL
LIN {X 0,Y 481.899,Z 577.524,A -85,B 0,C 180,E1 14205.889,E2 14205.889} C_VEL
LIN {X 0,Y 482.038,Z 578.102,A -85,B 0,C 180,E1 14205.787,E2 14205.787} C_VEL
LIN {X 0,Y 461.258,Z 800.045,A -85,B 0,C 180,E1 14202.472,E2 14202.472} C_VEL
LIN {X 0,Y 458.177,Z 824.001,A -85,B 0,C 180,E1 14202.075,E2 14202.075} C_VEL
LIN {X 0,Y 454.371,Z 845.703,A -85,B 0,C 180,E1 14201.64,E2 14201.64} C_VEL
LIN {X 0,Y 449.51,Z 868.005,A -85,B 0,C 180,E1 14201.078,E2 14201.078} C_VEL
LIN {X 0,Y 442.475,Z 894.453,A -85,B 0,C 180,E1 14200.247,E2 14200.247} C_VEL
LIN {X 0,Y 434.946,Z 917.836,A -85,B 0,C 180,E1 14199.327,E2 14199.327} C_VEL
LIN {X 0,Y 427.52,Z 938.113,A -85,B 0,C 180,E1 14198.38,E2 14198.38} C_VEL
LIN {X 0,Y 419.451,Z 957.852,A -85,B 0,C 180,E1 14197.294,E2 14197.294} C_VEL
LIN {X 0,Y 409.656,Z 979.466,A -85,B 0,C 180,E1 14195.899,E2 14195.899} C_VEL
LIN {X 0,Y 397.646,Z 1003.07,A -85,B 0,C 180,E1 14194.054,E2 14194.054} C_VEL
LIN {X 0,Y 387.755,Z 1020.855,A -85,B 0,C 180,E1 14192.398,E2 14192.398} C_VEL
LIN {X 0,Y 378.025,Z 1037.179,A -85,B 0,C 180,E1 14190.634,E2 14190.634} C_VEL
LIN {X 0,Y 368.101,Z 1052.821,A -85,B 0,C 180,E1 14188.678,E2 14188.678} C_VEL
LIN {X 0,Y 356.458,Z 1070.205,A -85,B 0,C 180,E1 14186.127,E2 14186.127} C_VEL
LIN {X 0,Y 343.519,Z 1088.323,A -85,B 0,C 180,E1 14182.893,E2 14182.893} C_VEL
LIN {X 0,Y 333.716,Z 1101.491,A -85,B 0,C 180,E1 14180.086,E2 14180.086} C_VEL
LIN {X 0,Y 324.569,Z 1113.483,A -85,B 0,C 180,E1 14177.091,E2 14177.091} C_VEL
LIN {X 0,Y 315.89,Z 1124.704,A -85,B 0,C 180,E1 14173.805,E2 14173.805} C_VEL
LIN {X 0,Y 306.052,Z 1137.517,A -85,B 0,C 180,E1 14169.33,E2 14169.33} C_VEL
LIN {X 0,Y 297.795,Z 1148.347,A -85,B 0,C 180,E1 14164.571,E2 14164.571} C_VEL
LIN {X 0,Y 292.182,Z 1156.178,A -85,B 0,C 180,E1 14160.414,E2 14160.414} C_VEL
LIN {X 0,Y 287.79,Z 1162.807,A -85,B 0,C 180,E1 14156.182,E2 14156.182} C_VEL
LIN {X 0,Y 284.253,Z 1168.844,A -85,B 0,C 180,E1 14151.458,E2 14151.458} C_VEL
LIN {X 0,Y 281.606,Z 1174.454,A -85,B 0,C 180,E1 14145.655,E2 14145.655} C_VEL
LIN {X 0,Y 280.522,Z 1177.669,A -85,B 0,C 180,E1 14140.889,E2 14140.889} C_VEL
LIN {X 0,Y 280.135,Z 1179.538,A -85,B 0,C 180,E1 14136.764,E2 14136.764} C_VEL
LIN {X 0,Y 280.009,Z 1180.538,A -85,B 0,C 180,E1 14132.661,E2 14132.661} C_VEL
LIN {X 0,Y 280.003,Z 1180.701,A -85,B 0,C 180,E1 14128.772,E2 14128.772} C_VEL
LIN {X 0,Y 280.062,Z 1180.027,A -85,B 0,C 180,E1 14124.674,E2 14124.674} C_VEL
LIN {X 0,Y 280.355,Z 1178.378,A -85,B 0,C 180,E1 14120.351,E2 14120.351} C_VEL
LIN {X 0,Y 281.106,Z 1175.759,A -85,B 0,C 180,E1 14116.003,E2 14116.003} C_VEL
LIN {X 0,Y 282.589,Z 1172.143,A -85,B 0,C 180,E1 14111.645,E2 14111.645} C_VEL
LIN {X 0,Y 284.994,Z 1167.497,A -85,B 0,C 180,E1 14107.299,E2 14107.299} C_VEL
LIN {X 0,Y 288.652,Z 1161.491,A -85,B 0,C 180,E1 14102.791,E2 14102.791} C_VEL
LIN {X 0,Y 294.624,Z 1152.881,A -85,B 0,C 180,E1 14097.575,E2 14097.575} C_VEL
LIN {X 0,Y 302.083,Z 1142.66,A -85,B 0,C 180,E1 14092.72,E2 14092.72} C_VEL
LIN {X 0,Y 309.318,Z 1133.234,A -85,B 0,C 180,E1 14088.99,E2 14088.99} C_VEL
LIN {X 0,Y 317.605,Z 1122.552,A -85,B 0,C 180,E1 14085.41,E2 14085.41} C_VEL
LIN {X 0,Y 328.443,Z 1108.645,A -85,B 0,C 180,E1 14081.507,E2 14081.507} C_VEL
LIN {X 0,Y 340.417,Z 1092.645,A -85,B 0,C 180,E1 14077.871,E2 14077.871} C_VEL
LIN {X 0,Y 350.26,Z 1079.068,A -85,B 0,C 180,E1 14075.272,E2 14075.272} C_VEL
LIN {X 0,Y 359.967,Z 1065.144,A -85,B 0,C 180,E1 14072.982,E2 14072.982} C_VEL
LIN {X 0,Y 370.519,Z 1049.267,A -85,B 0,C 180,E1 14070.742,E2 14070.742} C_VEL
LIN {X 0,Y 383.263,Z 1028.876,A -85,B 0,C 180,E1 14068.317,E2 14068.317} C_VEL
LIN {X 0,Y 395,Z 1008.197,A -85,B 0,C 180,E1 14066.295,E2 14066.295} C_VEL
LIN {X 0,Y 404.312,Z 990.523,A -85,B 0,C 180,E1 14064.827,E2 14064.827} C_VEL
LIN {X 0,Y 412.87,Z 972.873,A -85,B 0,C 180,E1 14063.553,E2 14063.553} C_VEL
LIN {X 0,Y 416.134,Z 965.951,A -85,B 0,C 180,E1 14063.099,E2 14063.099} C_VEL
LIN {X 0,Y 418.625,Z 959.665,A -85,B 0,C 180,E1 14062.574,E2 14062.574} C_VEL
LIN {X 0,Y 423.121,Z 943.237,A -85,B 0,C 180,E1 14060.85,E2 14060.85} C_VEL
LIN {X 0,Y 425.088,Z 937.568,A -85,B 0,C 180,E1 14060.465,E2 14060.465} C_VEL
LIN {X 0,Y 433.209,Z 915.651,A -85,B 0,C 180,E1 14059.468,E2 14059.468} C_VEL
LIN {X 0,Y 441.896,Z 888.077,A -85,B 0,C 180,E1 14058.447,E2 14058.447} C_VEL
LIN {X 0,Y 447.762,Z 865.663,A -85,B 0,C 180,E1 14057.78,E2 14057.78} C_VEL
LIN {X 0,Y 452.435,Z 844.217,A -85,B 0,C 180,E1 14057.259,E2 14057.259} C_VEL
LIN {X 0,Y 456.428,Z 821.307,A -85,B 0,C 180,E1 14056.818,E2 14056.818} C_VEL
LIN {X 0,Y 460.396,Z 787.319,A -85,B 0,C 180,E1 14056.28,E2 14056.28} C_VEL
LIN {X 0,Y 479.795,Z 583.813,A -85,B 0,C 180,E1 14053.266,E2 14053.266} C_VEL
LIN {X 0,Y 476.176,Z 577.204,A -85,B 0,C 180,E1 14050.71,E2 14050.71} C_VEL
LIN {X 0,Y 473.81,Z 573.002,A -85,B 0,C 180,E1 14048.617,E2 14048.617} C_VEL
LIN {X 0,Y 471.68,Z 569.048,A -85,B 0,C 180,E1 14046.084,E2 14046.084} C_VEL
LIN {X 0,Y 469.87,Z 564.912,A -85,B 0,C 180,E1 14041.707,E2 14041.707} C_VEL
LIN {X 0,Y 469.82,Z 564.357,A -85,B 0,C 180,E1 14040.976,E2 14040.976} C_VEL
LIN {X 0,Y 469.862,Z 564.662,A -85,B 0,C 180,E1 14038.903,E2 14038.903} C_VEL
LIN {X 0,Y 471.37,Z 568.693,A -85,B 0,C 180,E1 14034.767,E2 14034.767} C_VEL
LIN {X 0,Y 472.162,Z 569.894,A -85,B 0,C 180,E1 14033.678,E2 14033.678} C_VEL
LIN {X 0,Y 474.817,Z 574.772,A -85,B 0,C 180,E1 14030.852,E2 14030.852} C_VEL
LIN {X 0,Y 477.163,Z 579.048,A -85,B 0,C 180,E1 14028.946,E2 14028.946} C_VEL
LIN {X 0,Y 479.191,Z 582.885,A -85,B 0,C 180,E1 14027.528,E2 14027.528} C_VEL
LIN {X 0,Y 479.904,Z 584.786,A -85,B 0,C 180,E1 14027.032,E2 14027.032} C_VEL
LIN {X 0,Y 458.929,Z 805.58,A -85,B 0,C 180,E1 14023.756,E2 14023.756} C_VEL
LIN {X 0,Y 455.547,Z 832.16,A -85,B 0,C 180,E1 14023.318,E2 14023.318} C_VEL
LIN {X 0,Y 451.561,Z 854.449,A -85,B 0,C 180,E1 14022.903,E2 14022.903} C_VEL
LIN {X 0,Y 446.508,Z 876.864,A -85,B 0,C 180,E1 14022.402,E2 14022.402} C_VEL
LIN {X 0,Y 439.285,Z 903.363,A -85,B 0,C 180,E1 14021.646,E2 14021.646} C_VEL
LIN {X 0,Y 431.4,Z 927.23,A -85,B 0,C 180,E1 14020.784,E2 14020.784} C_VEL
LIN {X 0,Y 423.764,Z 947.636,A -85,B 0,C 180,E1 14019.895,E2 14019.895} C_VEL
LIN {X 0,Y 415.789,Z 966.797,A -85,B 0,C 180,E1 14018.912,E2 14018.912} C_VEL
LIN {X 0,Y 406.8,Z 986.44,A -85,B 0,C 180,E1 14017.726,E2 14017.726} C_VEL
LIN {X 0,Y 394.974,Z 1009.924,A -85,B 0,C 180,E1 14016.043,E2 14016.043} C_VEL
LIN {X 0,Y 382.759,Z 1031.627,A -85,B 0,C 180,E1 14014.135,E2 14014.135} C_VEL
LIN {X 0,Y 372.461,Z 1048.702,A -85,B 0,C 180,E1 14012.359,E2 14012.359} C_VEL
LIN {X 0,Y 361.947,Z 1065.123,A -85,B 0,C 180,E1 14010.363,E2 14010.363} C_VEL
LIN {X 0,Y 350.117,Z 1082.644,A -85,B 0,C 180,E1 14007.859,E2 14007.859} C_VEL
LIN {X 0,Y 336.38,Z 1101.754,A -85,B 0,C 180,E1 14004.532,E2 14004.532} C_VEL
LIN {X 0,Y 326.243,Z 1115.359,A -85,B 0,C 180,E1 14001.681,E2 14001.681} C_VEL
LIN {X 0,Y 316.904,Z 1127.633,A -85,B 0,C 180,E1 13998.669,E2 13998.669} C_VEL
LIN {X 0,Y 307.44,Z 1139.957,A -85,B 0,C 180,E1 13995.109,E2 13995.109} C_VEL
LIN {X 0,Y 297.349,Z 1153.304,A -85,B 0,C 180,E1 13990.464,E2 13990.464} C_VEL
LIN {X 0,Y 289.241,Z 1164.217,A -85,B 0,C 180,E1 13985.747,E2 13985.747} C_VEL
LIN {X 0,Y 283.485,Z 1172.575,A -85,B 0,C 180,E1 13981.398,E2 13981.398} C_VEL
LIN {X 0,Y 279.13,Z 1179.532,A -85,B 0,C 180,E1 13977.06,E2 13977.06} C_VEL
LIN {X 0,Y 275.666,Z 1185.981,A -85,B 0,C 180,E1 13972.161,E2 13972.161} C_VEL
LIN {X 0,Y 273.169,Z 1192.014,A -85,B 0,C 180,E1 13966.151,E2 13966.151} C_VEL
LIN {X 0,Y 272.244,Z 1195.509,A -85,B 0,C 180,E1 13961.224,E2 13961.224} C_VEL
LIN {X 0,Y 272.012,Z 1197.551,A -85,B 0,C 180,E1 13956.967,E2 13956.967} C_VEL
LIN {X 0,Y 271.997,Z 1198.619,A -85,B 0,C 180,E1 13952.95,E2 13952.95} C_VEL
LIN {X 0,Y 272.004,Z 1198.809,A -85,B 0,C 180,E1 13948.736,E2 13948.736} C_VEL
LIN {X 0,Y 271.992,Z 1198.046,A -85,B 0,C 180,E1 13944.515,E2 13944.515} C_VEL
LIN {X 0,Y 272.123,Z 1196.333,A -85,B 0,C 180,E1 13940.269,E2 13940.269} C_VEL
LIN {X 0,Y 272.697,Z 1193.501,A -85,B 0,C 180,E1 13935.779,E2 13935.779} C_VEL
LIN {X 0,Y 274.01,Z 1189.61,A -85,B 0,C 180,E1 13931.27,E2 13931.27} C_VEL
LIN {X 0,Y 276.3,Z 1184.641,A -85,B 0,C 180,E1 13926.769,E2 13926.769} C_VEL
LIN {X 0,Y 279.692,Z 1178.563,A -85,B 0,C 180,E1 13922.307,E2 13922.307} C_VEL
LIN {X 0,Y 284.541,Z 1170.977,A -85,B 0,C 180,E1 13917.716,E2 13917.716} C_VEL
LIN {X 0,Y 292.747,Z 1159.375,A -85,B 0,C 180,E1 13912.064,E2 13912.064} C_VEL
LIN {X 0,Y 300.677,Z 1148.72,A -85,B 0,C 180,E1 13907.866,E2 13907.866} C_VEL
LIN {X 0,Y 308.851,Z 1138.046,A -85,B 0,C 180,E1 13904.32,E2 13904.32} C_VEL
LIN {X 0,Y 318.409,Z 1125.616,A -85,B 0,C 180,E1 13900.819,E2 13900.819} C_VEL
LIN {X 0,Y 330.898,Z 1109.152,A -85,B 0,C 180,E1 13896.965,E2 13896.965} C_VEL
LIN {X 0,Y 342.935,Z 1092.571,A -85,B 0,C 180,E1 13893.805,E2 13893.805} C_VEL
LIN {X 0,Y 353.61,Z 1077.349,A -85,B 0,C 180,E1 13891.359,E2 13891.359} C_VEL
LIN {X 0,Y 364.199,Z 1061.529,A -85,B 0,C 180,E1 13889.188,E2 13889.188} C_VEL
LIN {X 0,Y 377.056,Z 1041.223,A -85,B 0,C 180,E1 13886.835,E2 13886.835} C_VEL
LIN {X 0,Y 389.374,Z 1019.816,A -85,B 0,C 180,E1 13884.806,E2 13884.806} C_VEL
LIN {X 0,Y 399.141,Z 1001.51,A -85,B 0,C 180,E1 13883.334,E2 13883.334} C_VEL
LIN {X 0,Y 408.325,Z 982.892,A -85,B 0,C 180,E1 13882.055,E2 13882.055} C_VEL
LIN {X 0,Y 417.589,Z 962.342,A -85,B 0,C 180,E1 13880.854,E2 13880.854} C_VEL
LIN {X 0,Y 428.19,Z 935.759,A -85,B 0,C 180,E1 13879.575,E2 13879.575} C_VEL
LIN {X 0,Y 435.737,Z 913.916,A -85,B 0,C 180,E1 13878.725,E2 13878.725} C_VEL
LIN {X 0,Y 442.162,Z 892.613,A -85,B 0,C 180,E1 13878.035,E2 13878.035} C_VEL
LIN {X 0,Y 447.761,Z 870.966,A -85,B 0,C 180,E1 13877.463,E2 13877.463} C_VEL
LIN {X 0,Y 453.487,Z 844.05,A -85,B 0,C 180,E1 13876.9,E2 13876.9} C_VEL
LIN {X 0,Y 457.486,Z 816.647,A -85,B 0,C 180,E1 13876.427,E2 13876.427} C_VEL
LIN {X 0,Y 469.856,Z 687.322,A -85,B 0,C 180,E1 13874.488,E2 13874.488} C_VEL
LIN {X 0,Y 479.714,Z 584.33,A -85,B 0,C 180,E1 13872.948,E2 13872.948} C_VEL
LIN {X 0,Y 477.798,Z 580.374,A -85,B 0,C 180,E1 13871.651,E2 13871.651} C_VEL
LIN {X 0,Y 475.231,Z 575.74,A -85,B 0,C 180,E1 13869.69,E2 13869.69} C_VEL
LIN {X 0,Y 473.65,Z 572.914,A -85,B 0,C 180,E1 13868.253,E2 13868.253} C_VEL
LIN {X 0,Y 471.585,Z 569,A -85,B 0,C 180,E1 13865.841,E2 13865.841} C_VEL
LIN {X 0,Y 469.751,Z 565.385,A -85,B 0,C 180,E1 13862.074,E2 13862.074} C_VEL
LIN {X 0,Y 469.602,Z 564.323,A -85,B 0,C 180,E1 13860.976,E2 13860.976} C_VEL
LIN {X 0,Y 469.643,Z 564.557,A -85,B 0,C 180,E1 13858.17,E2 13858.17} C_VEL
LIN {X 0,Y 471.57,Z 568.997,A -85,B 0,C 180,E1 13853.67,E2 13853.67} C_VEL
LIN {X 0,Y 474.413,Z 574.266,A -85,B 0,C 180,E1 13850.519,E2 13850.519} C_VEL
LIN {X 0,Y 477.271,Z 579.461,A -85,B 0,C 180,E1 13848.214,E2 13848.214} C_VEL
LIN {X 0,Y 479.613,Z 583.735,A -85,B 0,C 180,E1 13846.635,E2 13846.635} C_VEL
LIN {X 0,Y 458.61,Z 802.942,A -85,B 0,C 180,E1 13843.384,E2 13843.384} C_VEL
LIN {X 0,Y 455.597,Z 825.414,A -85,B 0,C 180,E1 13843.012,E2 13843.012} C_VEL
LIN {X 0,Y 451.635,Z 847.376,A -85,B 0,C 180,E1 13842.574,E2 13842.574} C_VEL
LIN {X 0,Y 445.831,Z 873.137,A -85,B 0,C 180,E1 13841.918,E2 13841.918} C_VEL
LIN {X 0,Y 438.6,Z 898.558,A -85,B 0,C 180,E1 13841.094,E2 13841.094} C_VEL
LIN {X 0,Y 431.762,Z 919.232,A -85,B 0,C 180,E1 13840.28,E2 13840.28} C_VEL
LIN {X 0,Y 424.211,Z 939.383,A -85,B 0,C 180,E1 13839.345,E2 13839.345} C_VEL
LIN {X 0,Y 416.025,Z 958.956,A -85,B 0,C 180,E1 13838.276,E2 13838.276} C_VEL
LIN {X 0,Y 404.862,Z 982.932,A -85,B 0,C 180,E1 13836.724,E2 13836.724} C_VEL
LIN {X 0,Y 393.313,Z 1004.82,A -85,B 0,C 180,E1 13834.995,E2 13834.995} C_VEL
LIN {X 0,Y 383.542,Z 1021.939,A -85,B 0,C 180,E1 13833.401,E2 13833.401} C_VEL
LIN {X 0,Y 373.713,Z 1038.002,A -85,B 0,C 180,E1 13831.67,E2 13831.67} C_VEL
LIN {X 0,Y 362.886,Z 1054.595,A -85,B 0,C 180,E1 13829.588,E2 13829.588} C_VEL
LIN {X 0,Y 349.398,Z 1073.99,A -85,B 0,C 180,E1 13826.67,E2 13826.67} C_VEL
LIN {X 0,Y 337.987,Z 1089.356,A -85,B 0,C 180,E1 13823.863,E2 13823.863} C_VEL
LIN {X 0,Y 327.892,Z 1102.455,A -85,B 0,C 180,E1 13821.04,E2 13821.04} C_VEL
LIN {X 0,Y 318.491,Z 1114.333,A -85,B 0,C 180,E1 13818.032,E2 13818.032} C_VEL
LIN {X 0,Y 308.726,Z 1126.492,A -85,B 0,C 180,E1 13814.391,E2 13814.391} C_VEL
LIN {X 0,Y 297.763,Z 1140.036,A -85,B 0,C 180,E1 13809.393,E2 13809.393} C_VEL
LIN {X 0,Y 290.664,Z 1149.016,A -85,B 0,C 180,E1 13805.303,E2 13805.303} C_VEL
LIN {X 0,Y 284.798,Z 1156.792,A -85,B 0,C 180,E1 13801.057,E2 13801.057} C_VEL
LIN {X 0,Y 280.005,Z 1163.667,A -85,B 0,C 180,E1 13796.51,E2 13796.51} C_VEL
LIN {X 0,Y 275.797,Z 1170.612,A -85,B 0,C 180,E1 13790.711,E2 13790.711} C_VEL
LIN {X 0,Y 273.55,Z 1175.181,A -85,B 0,C 180,E1 13785.475,E2 13785.475} C_VEL
LIN {X 0,Y 272.544,Z 1178.043,A -85,B 0,C 180,E1 13780.998,E2 13780.998} C_VEL
LIN {X 0,Y 272.141,Z 1179.866,A -85,B 0,C 180,E1 13776.752,E2 13776.752} C_VEL
LIN {X 0,Y 272.014,Z 1180.801,A -85,B 0,C 180,E1 13772.739,E2 13772.739} C_VEL
LIN {X 0,Y 272.007,Z 1180.964,A -85,B 0,C 180,E1 13768.736,E2 13768.736} C_VEL
LIN {X 0,Y 272.073,Z 1180.29,A -85,B 0,C 180,E1 13764.517,E2 13764.517} C_VEL
LIN {X 0,Y 272.394,Z 1178.643,A -85,B 0,C 180,E1 13760.066,E2 13760.066} C_VEL
LIN {X 0,Y 273.217,Z 1176.026,A -85,B 0,C 180,E1 13755.591,E2 13755.591} C_VEL
LIN {X 0,Y 274.833,Z 1172.379,A -85,B 0,C 180,E1 13751.073,E2 13751.073} C_VEL
LIN {X 0,Y 277.404,Z 1167.766,A -85,B 0,C 180,E1 13746.642,E2 13746.642} C_VEL
LIN {X 0,Y 281.1,Z 1162.055,A -85,B 0,C 180,E1 13742.228,E2 13742.228} C_VEL
LIN {X 0,Y 287.102,Z 1153.828,A -85,B 0,C 180,E1 13737.07,E2 13737.07} C_VEL
LIN {X 0,Y 295.144,Z 1143.38,A -85,B 0,C 180,E1 13731.935,E2 13731.935} C_VEL
LIN {X 0,Y 303.136,Z 1133.407,A -85,B 0,C 180,E1 13727.916,E2 13727.916} C_VEL
LIN {X 0,Y 311.71,Z 1122.824,A -85,B 0,C 180,E1 13724.332,E2 13724.332} C_VEL
LIN {X 0,Y 322.981,Z 1108.916,A -85,B 0,C 180,E1 13720.4,E2 13720.4} C_VEL
LIN {X 0,Y 334.944,Z 1093.492,A -85,B 0,C 180,E1 13716.868,E2 13716.868} C_VEL
LIN {X 0,Y 345.539,Z 1079.338,A -85,B 0,C 180,E1 13714.15,E2 13714.15} C_VEL
LIN {X 0,Y 356.176,Z 1064.499,A -85,B 0,C 180,E1 13711.725,E2 13711.725} C_VEL
LIN {X 0,Y 368.063,Z 1047.032,A -85,B 0,C 180,E1 13709.307,E2 13709.307} C_VEL
LIN {X 0,Y 381.583,Z 1025.472,A -85,B 0,C 180,E1 13706.848,E2 13706.848} C_VEL
LIN {X 0,Y 392.039,Z 1007.377,A -85,B 0,C 180,E1 13705.124,E2 13705.124} C_VEL
LIN {X 0,Y 402.046,Z 988.656,A -85,B 0,C 180,E1 13703.604,E2 13703.604} C_VEL
LIN {X 0,Y 411.983,Z 968.351,A -85,B 0,C 180,E1 13702.2,E2 13702.2} C_VEL
LIN {X 0,Y 422.866,Z 943.194,A -85,B 0,C 180,E1 13700.748,E2 13700.748} C_VEL
LIN {X 0,Y 425.088,Z 937.568,A -85,B 0,C 180,E1 13700.465,E2 13700.465} C_VEL
LIN {X 0,Y 427.429,Z 930.934,A -85,B 0,C 180,E1 13700.018,E2 13700.018} C_VEL
LIN {X 0,Y 431.397,Z 914.664,A -85,B 0,C 180,E1 13698.529,E2 13698.529} C_VEL
LIN {X 0,Y 433.36,Z 907.785,A -85,B 0,C 180,E1 13698.135,E2 13698.135} C_VEL
LIN {X 0,Y 440.035,Z 886.122,A -85,B 0,C 180,E1 13697.383,E2 13697.383} C_VEL
LIN {X 0,Y 445.635,Z 864.835,A -85,B 0,C 180,E1 13696.767,E2 13696.767} C_VEL
LIN {X 0,Y 450.384,Z 843.166,A -85,B 0,C 180,E1 13696.258,E2 13696.258} C_VEL
LIN {X 0,Y 454.987,Z 816.534,A -85,B 0,C 180,E1 13695.764,E2 13695.764} C_VEL
LIN {X 0,Y 459.39,Z 775.231,A -85,B 0,C 180,E1 13695.136,E2 13695.136} C_VEL
LIN {X 0,Y 477.446,Z 589.633,A -85,B 0,C 180,E1 13692.402,E2 13692.402} C_VEL
LIN {X 0,Y 474.303,Z 583.953,A -85,B 0,C 180,E1 13690.016,E2 13690.016} C_VEL
LIN {X 0,Y 472.584,Z 580.718,A -85,B 0,C 180,E1 13688.395,E2 13688.395} C_VEL
LIN {X 0,Y 470.616,Z 576.932,A -85,B 0,C 180,E1 13685.976,E2 13685.976} C_VEL
LIN {X 0,Y 468.873,Z 572.643,A -85,B 0,C 180,E1 13681.466,E2 13681.466} C_VEL
LIN {X 0,Y 468.799,Z 572.326,A -85,B 0,C 180,E1 13680.244,E2 13680.244} C_VEL
LIN {X 0,Y 468.873,Z 572.541,A -85,B 0,C 180,E1 13679.022,E2 13679.022} C_VEL
LIN {X 0,Y 470.312,Z 576.576,A -85,B 0,C 180,E1 13674.877,E2 13674.877} C_VEL
LIN {X 0,Y 471.041,Z 577.697,A -85,B 0,C 180,E1 13673.846,E2 13673.846} C_VEL
LIN {X 0,Y 473.627,Z 582.59,A -85,B 0,C 180,E1 13671.012,E2 13671.012} C_VEL
LIN {X 0,Y 475.927,Z 586.894,A -85,B 0,C 180,E1 13669.101,E2 13669.101} C_VEL
LIN {X 0,Y 477.604,Z 590.114,A -85,B 0,C 180,E1 13667.894,E2 13667.894} C_VEL
LIN {X 0,Y 456.592,Z 806.625,A -85,B 0,C 180,E1 13664.705,E2 13664.705} C_VEL
LIN {X 0,Y 453.275,Z 832.074,A -85,B 0,C 180,E1 13664.29,E2 13664.29} C_VEL
LIN {X 0,Y 449.248,Z 854.259,A -85,B 0,C 180,E1 13663.883,E2 13663.883} C_VEL
LIN {X 0,Y 444.106,Z 876.728,A -85,B 0,C 180,E1 13663.391,E2 13663.391} C_VEL
LIN {X 0,Y 436.803,Z 903.105,A -85,B 0,C 180,E1 13662.654,E2 13662.654} C_VEL
LIN {X 0,Y 428.505,Z 927.756,A -85,B 0,C 180,E1 13661.779,E2 13661.779} C_VEL
LIN {X 0,Y 421.03,Z 947.375,A -85,B 0,C 180,E1 13660.937,E2 13660.937} C_VEL
LIN {X 0,Y 412.914,Z 966.534,A -85,B 0,C 180,E1 13659.972,E2 13659.972} C_VEL
LIN {X 0,Y 403.718,Z 986.249,A -85,B 0,C 180,E1 13658.801,E2 13658.801} C_VEL
LIN {X 0,Y 391.692,Z 1009.657,A -85,B 0,C 180,E1 13657.148,E2 13657.148} C_VEL
LIN {X 0,Y 379.239,Z 1031.315,A -85,B 0,C 180,E1 13655.267,E2 13655.267} C_VEL
LIN {X 0,Y 368.315,Z 1048.993,A -85,B 0,C 180,E1 13653.442,E2 13653.442} C_VEL
LIN {X 0,Y 357.448,Z 1065.511,A -85,B 0,C 180,E1 13651.441,E2 13651.441} C_VEL
LIN {X 0,Y 343.928,Z 1084.925,A -85,B 0,C 180,E1 13648.641,E2 13648.641} C_VEL
LIN {X 0,Y 330.963,Z 1102.264,A -85,B 0,C 180,E1 13645.563,E2 13645.563} C_VEL
LIN {X 0,Y 320.52,Z 1115.797,A -85,B 0,C 180,E1 13642.699,E2 13642.699} C_VEL
LIN {X 0,Y 310.362,Z 1128.652,A -85,B 0,C 180,E1 13639.49,E2 13639.49} C_VEL
LIN {X 0,Y 298.896,Z 1143.088,A -85,B 0,C 180,E1 13635.168,E2 13635.168} C_VEL
LIN {X 0,Y 288.67,Z 1155.851,A -85,B 0,C 180,E1 13630.369,E2 13630.369} C_VEL
LIN {X 0,Y 281.808,Z 1164.775,A -85,B 0,C 180,E1 13626.336,E2 13626.336} C_VEL
LIN {X 0,Y 275.919,Z 1172.923,A -85,B 0,C 180,E1 13621.942,E2 13621.942} C_VEL
LIN {X 0,Y 270.772,Z 1180.823,A -85,B 0,C 180,E1 13616.776,E2 13616.776} C_VEL
LIN {X 0,Y 266.91,Z 1187.853,A -85,B 0,C 180,E1 13610.847,E2 13610.847} C_VEL
LIN {X 0,Y 265.082,Z 1192.327,A -85,B 0,C 180,E1 13605.874,E2 13605.874} C_VEL
LIN {X 0,Y 264.255,Z 1195.362,A -85,B 0,C 180,E1 13601.347,E2 13601.347} C_VEL
LIN {X 0,Y 264.018,Z 1197.301,A -85,B 0,C 180,E1 13597.136,E2 13597.136} C_VEL
LIN {X 0,Y 263.999,Z 1198.356,A -85,B 0,C 180,E1 13593.039,E2 13593.039} C_VEL
LIN {X 0,Y 264.007,Z 1198.569,A -85,B 0,C 180,E1 13588.915,E2 13588.915} C_VEL
LIN {X 0,Y 263.994,Z 1197.853,A -85,B 0,C 180,E1 13584.567,E2 13584.567} C_VEL
LIN {X 0,Y 264.144,Z 1196.067,A -85,B 0,C 180,E1 13579.972,E2 13579.972} C_VEL
LIN {X 0,Y 264.784,Z 1193.232,A -85,B 0,C 180,E1 13575.345,E2 13575.345} C_VEL
LIN {X 0,Y 266.219,Z 1189.339,A -85,B 0,C 180,E1 13570.7,E2 13570.7} C_VEL
LIN {X 0,Y 268.68,Z 1184.367,A -85,B 0,C 180,E1 13566.069,E2 13566.069} C_VEL
LIN {X 0,Y 272.309,Z 1178.287,A -85,B 0,C 180,E1 13561.489,E2 13561.489} C_VEL
LIN {X 0,Y 277.733,Z 1170.335,A -85,B 0,C 180,E1 13556.578,E2 13556.578} C_VEL
LIN {X 0,Y 286.477,Z 1158.626,A -85,B 0,C 180,E1 13550.823,E2 13550.823} C_VEL
LIN {X 0,Y 294.576,Z 1148.305,A -85,B 0,C 180,E1 13546.715,E2 13546.715} C_VEL
LIN {X 0,Y 303.009,Z 1137.767,A -85,B 0,C 180,E1 13543.177,E2 13543.177} C_VEL
LIN {X 0,Y 312.554,Z 1125.83,A -85,B 0,C 180,E1 13539.779,E2 13539.779} C_VEL
LIN {X 0,Y 325.253,Z 1109.742,A -85,B 0,C 180,E1 13535.957,E2 13535.957} C_VEL
LIN {X 0,Y 337.7,Z 1093.151,A -85,B 0,C 180,E1 13532.769,E2 13532.769} C_VEL
LIN {X 0,Y 348.734,Z 1077.899,A -85,B 0,C 180,E1 13530.307,E2 13530.307} C_VEL
LIN {X 0,Y 359.504,Z 1062.278,A -85,B 0,C 180,E1 13528.159,E2 13528.159} C_VEL
LIN {X 0,Y 370.352,Z 1045.625,A -85,B 0,C 180,E1 13526.202,E2 13526.202} C_VEL
LIN {X 0,Y 383.72,Z 1023.586,A -85,B 0,C 180,E1 13524.035,E2 13524.035} C_VEL
LIN {X 0,Y 395.135,Z 1002.791,A -85,B 0,C 180,E1 13522.352,E2 13522.352} C_VEL
LIN {X 0,Y 404.916,Z 983.435,A -85,B 0,C 180,E1 13521.03,E2 13521.03} C_VEL
LIN {X 0,Y 413.703,Z 964.406,A -85,B 0,C 180,E1 13519.923,E2 13519.923} C_VEL
LIN {X 0,Y 423.065,Z 941.965,A -85,B 0,C 180,E1 13518.822,E2 13518.822} C_VEL
LIN {X 0,Y 432.589,Z 915.538,A -85,B 0,C 180,E1 13517.774,E2 13517.774} C_VEL
LIN {X 0,Y 439.318,Z 893.774,A -85,B 0,C 180,E1 13517.074,E2 13517.074} C_VEL
LIN {X 0,Y 444.98,Z 872.431,A -85,B 0,C 180,E1 13516.513,E2 13516.513} C_VEL
LIN {X 0,Y 449.981,Z 849.803,A -85,B 0,C 180,E1 13516.038,E2 13516.038} C_VEL
LIN {X 0,Y 454.774,Z 820.66,A -85,B 0,C 180,E1 13515.523,E2 13515.523} C_VEL
LIN {X 0,Y 459.885,Z 770.498,A -85,B 0,C 180,E1 13514.764,E2 13514.764} C_VEL
LIN {X 0,Y 477.41,Z 589.971,A -85,B 0,C 180,E1 13512.107,E2 13512.107} C_VEL
LIN {X 0,Y 474.313,Z 584.04,A -85,B 0,C 180,E1 13509.77,E2 13509.77} C_VEL
LIN {X 0,Y 472.421,Z 580.625,A -85,B 0,C 180,E1 13508.03,E2 13508.03} C_VEL
LIN {X 0,Y 470.426,Z 576.783,A -85,B 0,C 180,E1 13505.611,E2 13505.611} C_VEL
LIN {X 0,Y 468.726,Z 573.114,A -85,B 0,C 180,E1 13501.834,E2 13501.834} C_VEL
LIN {X 0,Y 468.606,Z 572.266,A -85,B 0,C 180,E1 13500.856,E2 13500.856} C_VEL
LIN {X 0,Y 468.649,Z 572.439,A -85,B 0,C 180,E1 13498.288,E2 13498.288} C_VEL
LIN {X 0,Y 470.503,Z 576.881,A -85,B 0,C 180,E1 13493.778,E2 13493.778} C_VEL
LIN {X 0,Y 473.207,Z 582.05,A -85,B 0,C 180,E1 13490.698,E2 13490.698} C_VEL
LIN {X 0,Y 476.031,Z 587.303,A -85,B 0,C 180,E1 13488.367,E2 13488.367} C_VEL
LIN {X 0,Y 477.267,Z 589.641,A -85,B 0,C 180,E1 13487.488,E2 13487.488} C_VEL
LIN {X 0,Y 456.153,Z 805.213,A -85,B 0,C 180,E1 13484.317,E2 13484.317} C_VEL
LIN {X 0,Y 453.036,Z 827.474,A -85,B 0,C 180,E1 13483.949,E2 13483.949} C_VEL
LIN {X 0,Y 448.498,Z 851.677,A -85,B 0,C 180,E1 13483.459,E2 13483.459} C_VEL
LIN {X 0,Y 441.632,Z 879.804,A -85,B 0,C 180,E1 13482.716,E2 13482.716} C_VEL
LIN {X 0,Y 435.236,Z 901.385,A -85,B 0,C 180,E1 13482.003,E2 13482.003} C_VEL
LIN {X 0,Y 428.382,Z 921.504,A -85,B 0,C 180,E1 13481.21,E2 13481.21} C_VEL
LIN {X 0,Y 420.578,Z 941.764,A -85,B 0,C 180,E1 13480.27,E2 13480.27} C_VEL
LIN {X 0,Y 410.325,Z 965.523,A -85,B 0,C 180,E1 13478.95,E2 13478.95} C_VEL
LIN {X 0,Y 399.038,Z 988.249,A -85,B 0,C 180,E1 13477.419,E2 13477.419} C_VEL
LIN {X 0,Y 389.177,Z 1006.415,A -85,B 0,C 180,E1 13475.97,E2 13475.97} C_VEL
LIN {X 0,Y 379.107,Z 1023.589,A -85,B 0,C 180,E1 13474.37,E2 13474.37} C_VEL
LIN {X 0,Y 368.36,Z 1040.642,A -85,B 0,C 180,E1 13472.519,E2 13472.519} C_VEL
LIN {X 0,Y 354.491,Z 1061.064,A -85,B 0,C 180,E1 13469.863,E2 13469.863} C_VEL
LIN {X 0,Y 342.386,Z 1077.571,A -85,B 0,C 180,E1 13467.249,E2 13467.249} C_VEL
LIN {X 0,Y 331.959,Z 1091.147,A -85,B 0,C 180,E1 13464.711,E2 13464.711} C_VEL
LIN {X 0,Y 321.611,Z 1104.106,A -85,B 0,C 180,E1 13461.864,E2 13461.864} C_VEL
LIN {X 0,Y 310.527,Z 1117.622,A -85,B 0,C 180,E1 13458.332,E2 13458.332} C_VEL
LIN {X 0,Y 298.763,Z 1131.536,A -85,B 0,C 180,E1 13453.849,E2 13453.849} C_VEL
LIN {X 0,Y 290.219,Z 1141.652,A -85,B 0,C 180,E1 13449.852,E2 13449.852} C_VEL
LIN {X 0,Y 283.26,Z 1150.079,A -85,B 0,C 180,E1 13445.87,E2 13445.87} C_VEL
LIN {X 0,Y 277.205,Z 1157.733,A -85,B 0,C 180,E1 13441.534,E2 13441.534} C_VEL
LIN {X 0,Y 271.476,Z 1165.697,A -85,B 0,C 180,E1 13435.994,E2 13435.994} C_VEL
LIN {X 0,Y 267.523,Z 1171.855,A -85,B 0,C 180,E1 13430.259,E2 13430.259} C_VEL
LIN {X 0,Y 265.557,Z 1175.755,A -85,B 0,C 180,E1 13425.505,E2 13425.505} C_VEL
LIN {X 0,Y 264.567,Z 1178.417,A -85,B 0,C 180,E1 13421.113,E2 13421.113} C_VEL
LIN {X 0,Y 264.157,Z 1180.13,A -85,B 0,C 180,E1 13416.957,E2 13416.957} C_VEL
LIN {X 0,Y 264.02,Z 1181.064,A -85,B 0,C 180,E1 13412.822,E2 13412.822} C_VEL
LIN {X 0,Y 264.012,Z 1181.226,A -85,B 0,C 180,E1 13408.698,E2 13408.698} C_VEL
LIN {X 0,Y 264.085,Z 1180.553,A -85,B 0,C 180,E1 13404.351,E2 13404.351} C_VEL
LIN {X 0,Y 264.435,Z 1178.908,A -85,B 0,C 180,E1 13399.764,E2 13399.764} C_VEL
LIN {X 0,Y 265.339,Z 1176.293,A -85,B 0,C 180,E1 13395.153,E2 13395.153} C_VEL
LIN {X 0,Y 267.068,Z 1172.68,A -85,B 0,C 180,E1 13390.537,E2 13390.537} C_VEL
LIN {X 0,Y 269.849,Z 1168.036,A -85,B 0,C 180,E1 13385.947,E2 13385.947} C_VEL
LIN {X 0,Y 274.017,Z 1162.033,A -85,B 0,C 180,E1 13381.207,E2 13381.207} C_VEL
LIN {X 0,Y 280.751,Z 1153.361,A -85,B 0,C 180,E1 13375.717,E2 13375.717} C_VEL
LIN {X 0,Y 288.993,Z 1143.204,A -85,B 0,C 180,E1 13370.718,E2 13370.718} C_VEL
LIN {X 0,Y 296.9,Z 1133.779,A -85,B 0,C 180,E1 13366.872,E2 13366.872} C_VEL
LIN {X 0,Y 305.934,Z 1123.096,A -85,B 0,C 180,E1 13363.213,E2 13363.213} C_VEL
LIN {X 0,Y 317.674,Z 1109.155,A -85,B 0,C 180,E1 13359.246,E2 13359.246} C_VEL
LIN {X 0,Y 330.024,Z 1093.762,A -85,B 0,C 180,E1 13355.714,E2 13355.714} C_VEL
LIN {X 0,Y 340.955,Z 1079.607,A -85,B 0,C 180,E1 13352.997,E2 13352.997} C_VEL
LIN {X 0,Y 351.989,Z 1064.646,A -85,B 0,C 180,E1 13350.563,E2 13350.563} C_VEL
LIN {X 0,Y 364.451,Z 1046.799,A -85,B 0,C 180,E1 13348.113,E2 13348.113} C_VEL
LIN {X 0,Y 377.986,Z 1025.677,A -85,B 0,C 180,E1 13345.733,E2 13345.733} C_VEL
LIN {X 0,Y 388.636,Z 1007.641,A -85,B 0,C 180,E1 13344.032,E2 13344.032} C_VEL
LIN {X 0,Y 398.542,Z 989.499,A -85,B 0,C 180,E1 13342.573,E2 13342.573} C_VEL
LIN {X 0,Y 408.094,Z 970.426,A -85,B 0,C 180,E1 13341.261,E2 13341.261} C_VEL
LIN {X 0,Y 419.547,Z 944.752,A -85,B 0,C 180,E1 13339.781,E2 13339.781} C_VEL
LIN {X 0,Y 428.139,Z 922.649,A -85,B 0,C 180,E1 13338.74,E2 13338.74} C_VEL
LIN {X 0,Y 433.36,Z 907.785,A -85,B 0,C 180,E1 13338.135,E2 13338.135} C_VEL
LIN {X 0,Y 435.338,Z 900.824,A -85,B 0,C 180,E1 13337.759,E2 13337.759} C_VEL
LIN {X 0,Y 438.962,Z 882.804,A -85,B 0,C 180,E1 13336.367,E2 13336.367} C_VEL
LIN {X 0,Y 440.467,Z 876.709,A -85,B 0,C 180,E1 13336.087,E2 13336.087} C_VEL
LIN {X 0,Y 447.014,Z 849.262,A -85,B 0,C 180,E1 13335.398,E2 13335.398} C_VEL
LIN {X 0,Y 451.232,Z 826.818,A -85,B 0,C 180,E1 13334.961,E2 13334.961} C_VEL
LIN {X 0,Y 454.358,Z 804.575,A -85,B 0,C 180,E1 13334.6,E2 13334.6} C_VEL
LIN {X 0,Y 475.219,Z 595.721,A -85,B 0,C 180,E1 13331.557,E2 13331.557} C_VEL
LIN {X 0,Y 472.701,Z 591.025,A -85,B 0,C 180,E1 13329.497,E2 13329.497} C_VEL
LIN {X 0,Y 471.366,Z 588.432,A -85,B 0,C 180,E1 13328.171,E2 13328.171} C_VEL
LIN {X 0,Y 469.467,Z 584.725,A -85,B 0,C 180,E1 13325.745,E2 13325.745} C_VEL
LIN {X 0,Y 467.885,Z 580.524,A -85,B 0,C 180,E1 13321.347,E2 13321.347} C_VEL
LIN {X 0,Y 467.856,Z 580.293,A -85,B 0,C 180,E1 13319.51,E2 13319.51} C_VEL
LIN {X 0,Y 469.924,Z 585.5,A -85,B 0,C 180,E1 13314.015,E2 13314.015} C_VEL
LIN {X 0,Y 472.379,Z 590.277,A -85,B 0,C 180,E1 13311.234,E2 13311.234} C_VEL
LIN {X 0,Y 474.617,Z 594.588,A -85,B 0,C 180,E1 13309.316,E2 13309.316} C_VEL
LIN {X 0,Y 475.341,Z 596.232,A -85,B 0,C 180,E1 13308.749,E2 13308.749} C_VEL
LIN {X 0,Y 454.027,Z 810.654,A -85,B 0,C 180,E1 13305.618,E2 13305.618} C_VEL
LIN {X 0,Y 450.896,Z 833.454,A -85,B 0,C 180,E1 13305.246,E2 13305.246} C_VEL
LIN {X 0,Y 446.693,Z 855.868,A -85,B 0,C 180,E1 13304.839,E2 13304.839} C_VEL
LIN {X 0,Y 440.464,Z 882.181,A -85,B 0,C 180,E1 13304.256,E2 13304.256} C_VEL
LIN {X 0,Y 432.745,Z 908.008,A -85,B 0,C 180,E1 13303.507,E2 13303.507} C_VEL
LIN {X 0,Y 425.588,Z 928.696,A -85,B 0,C 180,E1 13302.771,E2 13302.771} C_VEL
LIN {X 0,Y 418.022,Z 948.124,A -85,B 0,C 180,E1 13301.947,E2 13301.947} C_VEL
LIN {X 0,Y 409.366,Z 968.084,A -85,B 0,C 180,E1 13300.949,E2 13300.949} C_VEL
LIN {X 0,Y 398.067,Z 991.636,A -85,B 0,C 180,E1 13299.536,E2 13299.536} C_VEL
LIN {X 0,Y 385.825,Z 1014.107,A -85,B 0,C 180,E1 13297.888,E2 13297.888} C_VEL
LIN {X 0,Y 375.087,Z 1032.276,A -85,B 0,C 180,E1 13296.299,E2 13296.299} C_VEL
LIN {X 0,Y 364.305,Z 1049.285,A -85,B 0,C 180,E1 13294.55,E2 13294.55} C_VEL
LIN {X 0,Y 352.729,Z 1066.408,A -85,B 0,C 180,E1 13292.48,E2 13292.48} C_VEL
LIN {X 0,Y 337.816,Z 1086.993,A -85,B 0,C 180,E1 13289.462,E2 13289.462} C_VEL
LIN {X 0,Y 325.905,Z 1102.46,A -85,B 0,C 180,E1 13286.689,E2 13286.689} C_VEL
LIN {X 0,Y 315.213,Z 1115.853,A -85,B 0,C 180,E1 13283.842,E2 13283.842} C_VEL
LIN {X 0,Y 304.947,Z 1128.377,A -85,B 0,C 180,E1 13280.696,E2 13280.696} C_VEL
LIN {X 0,Y 292.991,Z 1142.811,A -85,B 0,C 180,E1 13276.341,E2 13276.341} C_VEL
LIN {X 0,Y 282.292,Z 1155.576,A -85,B 0,C 180,E1 13271.478,E2 13271.478} C_VEL
LIN {X 0,Y 275.063,Z 1164.499,A -85,B 0,C 180,E1 13267.376,E2 13267.376} C_VEL
LIN {X 0,Y 269.092,Z 1172.284,A -85,B 0,C 180,E1 13263.107,E2 13263.107} C_VEL
LIN {X 0,Y 263.946,Z 1179.611,A -85,B 0,C 180,E1 13258.263,E2 13258.263} C_VEL
LIN {X 0,Y 259.443,Z 1187.151,A -85,B 0,C 180,E1 13251.952,E2 13251.952} C_VEL
LIN {X 0,Y 257.233,Z 1191.977,A -85,B 0,C 180,E1 13246.484,E2 13246.484} C_VEL
LIN {X 0,Y 256.287,Z 1195.105,A -85,B 0,C 180,E1 13241.687,E2 13241.687} C_VEL
LIN {X 0,Y 256.024,Z 1197.07,A -85,B 0,C 180,E1 13237.256,E2 13237.256} C_VEL
LIN {X 0,Y 256.002,Z 1198.094,A -85,B 0,C 180,E1 13233.134,E2 13233.134} C_VEL
LIN {X 0,Y 256.012,Z 1198.307,A -85,B 0,C 180,E1 13228.881,E2 13228.881} C_VEL
LIN {X 0,Y 255.998,Z 1197.589,A -85,B 0,C 180,E1 13224.397,E2 13224.397} C_VEL
LIN {X 0,Y 256.172,Z 1195.777,A -85,B 0,C 180,E1 13219.613,E2 13219.613} C_VEL
LIN {X 0,Y 256.886,Z 1192.949,A -85,B 0,C 180,E1 13214.864,E2 13214.864} C_VEL
LIN {X 0,Y 258.455,Z 1189.042,A -85,B 0,C 180,E1 13210.069,E2 13210.069} C_VEL
LIN {X 0,Y 261.098,Z 1184.093,A -85,B 0,C 180,E1 13205.329,E2 13205.329} C_VEL
LIN {X 0,Y 264.981,Z 1178.012,A -85,B 0,C 180,E1 13200.625,E2 13200.625} C_VEL
LIN {X 0,Y 270.752,Z 1170.058,A -85,B 0,C 180,E1 13195.597,E2 13195.597} C_VEL
LIN {X 0,Y 279.98,Z 1158.347,A -85,B 0,C 180,E1 13189.731,E2 13189.731} C_VEL
LIN {X 0,Y 288.507,Z 1148.004,A -85,B 0,C 180,E1 13185.557,E2 13185.557} C_VEL
LIN {X 0,Y 297.285,Z 1137.487,A -85,B 0,C 180,E1 13181.988,E2 13181.988} C_VEL
LIN {X 0,Y 307.623,Z 1125.057,A -85,B 0,C 180,E1 13178.435,E2 13178.435} C_VEL
LIN {X 0,Y 321.182,Z 1108.387,A -85,B 0,C 180,E1 13174.513,E2 13174.513} C_VEL
LIN {X 0,Y 333.864,Z 1092.013,A -85,B 0,C 180,E1 13171.404,E2 13171.404} C_VEL
LIN {X 0,Y 345.174,Z 1076.793,A -85,B 0,C 180,E1 13168.979,E2 13168.979} C_VEL
LIN {X 0,Y 356.7,Z 1060.46,A -85,B 0,C 180,E1 13166.776,E2 13166.776} C_VEL
LIN {X 0,Y 370.618,Z 1039.386,A -85,B 0,C 180,E1 13164.405,E2 13164.405} C_VEL
LIN {X 0,Y 383.106,Z 1018.589,A -85,B 0,C 180,E1 13162.498,E2 13162.498} C_VEL
LIN {X 0,Y 392.956,Z 1000.871,A -85,B 0,C 180,E1 13161.121,E2 13161.121} C_VEL
LIN {X 0,Y 402.443,Z 982.343,A -85,B 0,C 180,E1 13159.887,E2 13159.887} C_VEL
LIN {X 0,Y 412.222,Z 961.413,A -85,B 0,C 180,E1 13158.708,E2 13158.708} C_VEL
LIN {X 0,Y 423.014,Z 935.211,A -85,B 0,C 180,E1 13157.497,E2 13157.497} C_VEL
LIN {X 0,Y 431.026,Z 912.682,A -85,B 0,C 180,E1 13156.657,E2 13156.657} C_VEL
LIN {X 0,Y 437.52,Z 891.731,A -85,B 0,C 180,E1 13156.01,E2 13156.01} C_VEL
LIN {X 0,Y 443.295,Z 869.991,A -85,B 0,C 180,E1 13155.464,E2 13155.464} C_VEL
LIN {X 0,Y 449.204,Z 842.691,A -85,B 0,C 180,E1 13154.919,E2 13154.919} C_VEL
LIN {X 0,Y 453.218,Z 815.862,A -85,B 0,C 180,E1 13154.47,E2 13154.47} C_VEL
LIN {X 0,Y 468.809,Z 659.317,A -85,B 0,C 180,E1 13152.171,E2 13152.171} C_VEL
LIN {X 0,Y 475.145,Z 595.768,A -85,B 0,C 180,E1 13151.231,E2 13151.231} C_VEL
LIN {X 0,Y 472.559,Z 590.864,A -85,B 0,C 180,E1 13149.131,E2 13149.131} C_VEL
LIN {X 0,Y 471.082,Z 588.153,A -85,B 0,C 180,E1 13147.685,E2 13147.685} C_VEL
LIN {X 0,Y 469.362,Z 584.663,A -85,B 0,C 180,E1 13145.501,E2 13145.501} C_VEL
LIN {X 0,Y 467.723,Z 580.994,A -85,B 0,C 180,E1 13141.715,E2 13141.715} C_VEL
LIN {X 0,Y 467.632,Z 580.207,A -85,B 0,C 180,E1 13140.858,E2 13140.858} C_VEL
LIN {X 0,Y 467.657,Z 580.321,A -85,B 0,C 180,E1 13138.407,E2 13138.407} C_VEL
LIN {X 0,Y 469.725,Z 585.44,A -85,B 0,C 180,E1 13133.461,E2 13133.461} C_VEL
LIN {X 0,Y 472.025,Z 589.875,A -85,B 0,C 180,E1 13130.858,E2 13130.858} C_VEL
LIN {X 0,Y 474.714,Z 594.998,A -85,B 0,C 180,E1 13128.58,E2 13128.58} C_VEL
LIN {X 0,Y 475.008,Z 595.738,A -85,B 0,C 180,E1 13128.346,E2 13128.346} C_VEL
LIN {X 0,Y 453.889,Z 806.886,A -85,B 0,C 180,E1 13125.268,E2 13125.268} C_VEL
LIN {X 0,Y 450.518,Z 830.02,A -85,B 0,C 180,E1 13124.887,E2 13124.887} C_VEL
LIN {X 0,Y 444.799,Z 858.572,A -85,B 0,C 180,E1 13124.292,E2 13124.292} C_VEL
LIN {X 0,Y 438.679,Z 882.286,A -85,B 0,C 180,E1 13123.65,E2 13123.65} C_VEL
LIN {X 0,Y 432.399,Z 902.935,A -85,B 0,C 180,E1 13122.971,E2 13122.971} C_VEL
LIN {X 0,Y 425.348,Z 923.146,A -85,B 0,C 180,E1 13122.18,E2 13122.18} C_VEL
LIN {X 0,Y 416.339,Z 945.914,A -85,B 0,C 180,E1 13121.121,E2 13121.121} C_VEL
LIN {X 0,Y 405.074,Z 970.631,A -85,B 0,C 180,E1 13119.712,E2 13119.712} C_VEL
LIN {X 0,Y 395.587,Z 989.25,A -85,B 0,C 180,E1 13118.455,E2 13118.455} C_VEL
LIN {X 0,Y 385.538,Z 1007.349,A -85,B 0,C 180,E1 13117.022,E2 13117.022} C_VEL
LIN {X 0,Y 374.996,Z 1024.892,A -85,B 0,C 180,E1 13115.397,E2 13115.397} C_VEL
LIN {X 0,Y 361.888,Z 1045.124,A -85,B 0,C 180,E1 13113.178,E2 13113.178} C_VEL
LIN {X 0,Y 348.163,Z 1064.339,A -85,B 0,C 180,E1 13110.587,E2 13110.587} C_VEL
LIN {X 0,Y 337.325,Z 1078.678,A -85,B 0,C 180,E1 13108.287,E2 13108.287} C_VEL
LIN {X 0,Y 326.403,Z 1092.445,A -85,B 0,C 180,E1 13105.691,E2 13105.691} C_VEL
LIN {X 0,Y 314.834,Z 1106.446,A -85,B 0,C 180,E1 13102.556,E2 13102.556} C_VEL
LIN {X 0,Y 301.443,Z 1121.993,A -85,B 0,C 180,E1 13098.271,E2 13098.271} C_VEL
LIN {X 0,Y 291.443,Z 1133.321,A -85,B 0,C 180,E1 13094.416,E2 13094.416} C_VEL
LIN {X 0,Y 283.079,Z 1142.822,A -85,B 0,C 180,E1 13090.534,E2 13090.534} C_VEL
LIN {X 0,Y 275.23,Z 1151.929,A -85,B 0,C 180,E1 13086.052,E2 13086.052} C_VEL
LIN {X 0,Y 267.088,Z 1161.866,A -85,B 0,C 180,E1 13079.861,E2 13079.861} C_VEL
LIN {X 0,Y 262.554,Z 1167.957,A -85,B 0,C 180,E1 13074.989,E2 13074.989} C_VEL
LIN {X 0,Y 259.511,Z 1172.651,A -85,B 0,C 180,E1 13070.289,E2 13070.289} C_VEL
LIN {X 0,Y 257.627,Z 1176.195,A -85,B 0,C 180,E1 13065.734,E2 13065.734} C_VEL
LIN {X 0,Y 256.591,Z 1178.792,A -85,B 0,C 180,E1 13061.235,E2 13061.235} C_VEL
LIN {X 0,Y 256.162,Z 1180.459,A -85,B 0,C 180,E1 13056.95,E2 13056.95} C_VEL
LIN {X 0,Y 256.022,Z 1181.348,A -85,B 0,C 180,E1 13052.686,E2 13052.686} C_VEL
LIN {X 0,Y 256.017,Z 1181.467,A -85,B 0,C 180,E1 13048.433,E2 13048.433} C_VEL
LIN {X 0,Y 256.111,Z 1180.752,A -85,B 0,C 180,E1 13043.949,E2 13043.949} C_VEL
LIN {X 0,Y 256.482,Z 1179.173,A -85,B 0,C 180,E1 13039.443,E2 13039.443} C_VEL
LIN {X 0,Y 257.475,Z 1176.559,A -85,B 0,C 180,E1 13034.689,E2 13034.689} C_VEL
LIN {X 0,Y 259.348,Z 1172.948,A -85,B 0,C 180,E1 13029.933,E2 13029.933} C_VEL
LIN {X 0,Y 262.331,Z 1168.307,A -85,B 0,C 180,E1 13025.212,E2 13025.212} C_VEL
LIN {X 0,Y 266.665,Z 1162.44,A -85,B 0,C 180,E1 13020.449,E2 13020.449} C_VEL
LIN {X 0,Y 273.857,Z 1153.697,A -85,B 0,C 180,E1 13014.77,E2 13014.77} C_VEL
LIN {X 0,Y 282.573,Z 1143.477,A -85,B 0,C 180,E1 13009.645,E2 13009.645} C_VEL
LIN {X 0,Y 290.857,Z 1134.051,A -85,B 0,C 180,E1 13005.746,E2 13005.746} C_VEL
LIN {X 0,Y 300.282,Z 1123.368,A -85,B 0,C 180,E1 13002.053,E2 13002.053} C_VEL
LIN {X 0,Y 312.442,Z 1109.459,A -85,B 0,C 180,E1 12998.072,E2 12998.072} C_VEL
LIN {X 0,Y 325.241,Z 1094.032,A -85,B 0,C 180,E1 12994.525,E2 12994.525} C_VEL
LIN {X 0,Y 336.514,Z 1079.876,A -85,B 0,C 180,E1 12991.814,E2 12991.814} C_VEL
LIN {X 0,Y 347.395,Z 1065.539,A -85,B 0,C 180,E1 12989.484,E2 12989.484} C_VEL
LIN {X 0,Y 359.214,Z 1049.068,A -85,B 0,C 180,E1 12987.213,E2 12987.213} C_VEL
LIN {X 0,Y 374.09,Z 1026.604,A -85,B 0,C 180,E1 12984.668,E2 12984.668} C_VEL
LIN {X 0,Y 384.996,Z 1008.566,A -85,B 0,C 180,E1 12982.978,E2 12982.978} C_VEL
LIN {X 0,Y 395.171,Z 990.342,A -85,B 0,C 180,E1 12981.524,E2 12981.524} C_VEL
LIN {X 0,Y 404.519,Z 972.094,A -85,B 0,C 180,E1 12980.279,E2 12980.279} C_VEL
LIN {X 0,Y 415.38,Z 948.66,A -85,B 0,C 180,E1 12978.918,E2 12978.918} C_VEL
LIN {X 0,Y 425.201,Z 924.03,A -85,B 0,C 180,E1 12977.758,E2 12977.758} C_VEL
LIN {X 0,Y 432.568,Z 902.978,A -85,B 0,C 180,E1 12976.933,E2 12976.933} C_VEL
LIN {X 0,Y 438.54,Z 883.423,A -85,B 0,C 180,E1 12976.287,E2 12976.287} C_VEL
LIN {X 0,Y 440.467,Z 876.709,A -85,B 0,C 180,E1 12976.087,E2 12976.087} C_VEL
LIN {X 0,Y 442.153,Z 869.552,A -85,B 0,C 180,E1 12975.761,E2 12975.761} C_VEL
LIN {X 0,Y 444.725,Z 851.823,A -85,B 0,C 180,E1 12974.576,E2 12974.576} C_VEL
LIN {X 0,Y 445.99,Z 844.495,A -85,B 0,C 180,E1 12974.298,E2 12974.298} C_VEL
LIN {X 0,Y 450.314,Z 820.541,A -85,B 0,C 180,E1 12973.864,E2 12973.864} C_VEL
LIN {X 0,Y 454.573,Z 784.73,A -85,B 0,C 180,E1 12973.321,E2 12973.321} C_VEL
LIN {X 0,Y 473.07,Z 601.815,A -85,B 0,C 180,E1 12970.689,E2 12970.689} C_VEL
LIN {X 0,Y 470.27,Z 596.32,A -85,B 0,C 180,E1 12968.067,E2 12968.067} C_VEL
LIN {X 0,Y 468.408,Z 592.608,A -85,B 0,C 180,E1 12965.635,E2 12965.635} C_VEL
LIN {X 0,Y 466.899,Z 588.405,A -85,B 0,C 180,E1 12961.227,E2 12961.227} C_VEL
LIN {X 0,Y 466.902,Z 588.436,A -85,B 0,C 180,E1 12959.141,E2 12959.141} C_VEL
LIN {X 0,Y 468.281,Z 592.431,A -85,B 0,C 180,E1 12954.978,E2 12954.978} C_VEL
LIN {X 0,Y 468.931,Z 593.636,A -85,B 0,C 180,E1 12954.003,E2 12954.003} C_VEL
LIN {X 0,Y 471.198,Z 598.094,A -85,B 0,C 180,E1 12951.396,E2 12951.396} C_VEL
LIN {X 0,Y 473.209,Z 602.071,A -85,B 0,C 180,E1 12949.617,E2 12949.617} C_VEL
LIN {X 0,Y 451.854,Z 812.406,A -85,B 0,C 180,E1 12946.576,E2 12946.576} C_VEL
LIN {X 0,Y 448.656,Z 834.764,A -85,B 0,C 180,E1 12946.214,E2 12946.214} C_VEL
LIN {X 0,Y 443.902,Z 859.214,A -85,B 0,C 180,E1 12945.773,E2 12945.773} C_VEL
LIN {X 0,Y 436.829,Z 887.102,A -85,B 0,C 180,E1 12945.137,E2 12945.137} C_VEL
LIN {X 0,Y 429.961,Z 909.4,A -85,B 0,C 180,E1 12944.488,E2 12944.488} C_VEL
LIN {X 0,Y 422.782,Z 929.686,A -85,B 0,C 180,E1 12943.774,E2 12943.774} C_VEL
LIN {X 0,Y 414.724,Z 949.885,A -85,B 0,C 180,E1 12942.924,E2 12942.924} C_VEL
LIN {X 0,Y 404.286,Z 973.261,A -85,B 0,C 180,E1 12941.747,E2 12941.747} C_VEL
LIN {X 0,Y 392.42,Z 996.591,A -85,B 0,C 180,E1 12940.298,E2 12940.298} C_VEL
LIN {X 0,Y 381.998,Z 1015.188,A -85,B 0,C 180,E1 12938.926,E2 12938.926} C_VEL
LIN {X 0,Y 371.445,Z 1032.622,A -85,B 0,C 180,E1 12937.411,E2 12937.411} C_VEL
LIN {X 0,Y 360.251,Z 1049.851,A -85,B 0,C 180,E1 12935.651,E2 12935.651} C_VEL
LIN {X 0,Y 346.894,Z 1069.075,A -85,B 0,C 180,E1 12933.318,E2 12933.318} C_VEL
LIN {X 0,Y 332.271,Z 1088.436,A -85,B 0,C 180,E1 12930.417,E2 12930.417} C_VEL
LIN {X 0,Y 320.681,Z 1103.019,A -85,B 0,C 180,E1 12927.779,E2 12927.779} C_VEL
LIN {X 0,Y 309.64,Z 1116.379,A -85,B 0,C 180,E1 12924.914,E2 12924.914} C_VEL
LIN {X 0,Y 297.481,Z 1130.691,A -85,B 0,C 180,E1 12921.239,E2 12921.239} C_VEL
LIN {X 0,Y 284.823,Z 1145.173,A -85,B 0,C 180,E1 12916.607,E2 12916.607} C_VEL
LIN {X 0,Y 275.606,Z 1155.77,A -85,B 0,C 180,E1 12912.437,E2 12912.437} C_VEL
LIN {X 0,Y 268.065,Z 1164.64,A -85,B 0,C 180,E1 12908.255,E2 12908.255} C_VEL
LIN {X 0,Y 261.269,Z 1173.08,A -85,B 0,C 180,E1 12903.457,E2 12903.457} C_VEL
LIN {X 0,Y 254.786,Z 1181.999,A -85,B 0,C 180,E1 12897.079,E2 12897.079} C_VEL
LIN {X 0,Y 251.258,Z 1187.741,A -85,B 0,C 180,E1 12891.721,E2 12891.721} C_VEL
LIN {X 0,Y 249.302,Z 1191.876,A -85,B 0,C 180,E1 12886.784,E2 12886.784} C_VEL
LIN {X 0,Y 248.331,Z 1194.829,A -85,B 0,C 180,E1 12882.085,E2 12882.085} C_VEL
LIN {X 0,Y 248.039,Z 1196.759,A -85,B 0,C 180,E1 12877.644,E2 12877.644} C_VEL
LIN {X 0,Y 248.004,Z 1197.831,A -85,B 0,C 180,E1 12873.236,E2 12873.236} C_VEL
LIN {X 0,Y 248.016,Z 1198.044,A -85,B 0,C 180,E1 12868.845,E2 12868.845} C_VEL
LIN {X 0,Y 248.002,Z 1197.325,A -85,B 0,C 180,E1 12864.215,E2 12864.215} C_VEL
LIN {X 0,Y 248.194,Z 1195.534,A -85,B 0,C 180,E1 12859.321,E2 12859.321} C_VEL
LIN {X 0,Y 248.988,Z 1192.694,A -85,B 0,C 180,E1 12854.392,E2 12854.392} C_VEL
LIN {X 0,Y 250.686,Z 1188.796,A -85,B 0,C 180,E1 12849.452,E2 12849.452} C_VEL
LIN {X 0,Y 253.555,Z 1183.819,A -85,B 0,C 180,E1 12844.544,E2 12844.544} C_VEL
LIN {X 0,Y 257.712,Z 1177.736,A -85,B 0,C 180,E1 12839.711,E2 12839.711} C_VEL
LIN {X 0,Y 263.856,Z 1169.778,A -85,B 0,C 180,E1 12834.563,E2 12834.563} C_VEL
LIN {X 0,Y 273.594,Z 1158.069,A -85,B 0,C 180,E1 12828.588,E2 12828.588} C_VEL
LIN {X 0,Y 282.514,Z 1147.747,A -85,B 0,C 180,E1 12824.365,E2 12824.365} C_VEL
LIN {X 0,Y 291.688,Z 1137.208,A -85,B 0,C 180,E1 12820.751,E2 12820.751} C_VEL
LIN {X 0,Y 302.435,Z 1124.777,A -85,B 0,C 180,E1 12817.179,E2 12817.179} C_VEL
LIN {X 0,Y 316.054,Z 1108.648,A -85,B 0,C 180,E1 12813.365,E2 12813.365} C_VEL
LIN {X 0,Y 329.564,Z 1091.735,A -85,B 0,C 180,E1 12810.157,E2 12810.157} C_VEL
LIN {X 0,Y 341.19,Z 1076.515,A -85,B 0,C 180,E1 12807.748,E2 12807.748} C_VEL
LIN {X 0,Y 353.013,Z 1060.183,A -85,B 0,C 180,E1 12805.564,E2 12805.564} C_VEL
LIN {X 0,Y 366.952,Z 1039.609,A -85,B 0,C 180,E1 12803.273,E2 12803.273} C_VEL
LIN {X 0,Y 380.014,Z 1018.313,A -85,B 0,C 180,E1 12801.345,E2 12801.345} C_VEL
LIN {X 0,Y 389.976,Z 1000.759,A -85,B 0,C 180,E1 12800.004,E2 12800.004} C_VEL
LIN {X 0,Y 399.868,Z 981.786,A -85,B 0,C 180,E1 12798.763,E2 12798.763} C_VEL
LIN {X 0,Y 409.786,Z 960.894,A -85,B 0,C 180,E1 12797.612,E2 12797.612} C_VEL
LIN {X 0,Y 421.063,Z 933.8,A -85,B 0,C 180,E1 12796.396,E2 12796.396} C_VEL
LIN {X 0,Y 428.771,Z 912.408,A -85,B 0,C 180,E1 12795.618,E2 12795.618} C_VEL
LIN {X 0,Y 435.162,Z 892.129,A -85,B 0,C 180,E1 12795.005,E2 12795.005} C_VEL
LIN {X 0,Y 440.941,Z 870.793,A -85,B 0,C 180,E1 12794.478,E2 12794.478} C_VEL
LIN {X 0,Y 446.501,Z 845.917,A -85,B 0,C 180,E1 12793.986,E2 12793.986} C_VEL
LIN {X 0,Y 451.079,Z 817.188,A -85,B 0,C 180,E1 12793.504,E2 12793.504} C_VEL
LIN {X 0,Y 458.762,Z 742.601,A -85,B 0,C 180,E1 12792.409,E2 12792.409} C_VEL
LIN {X 0,Y 473.008,Z 601.909,A -85,B 0,C 180,E1 12790.385,E2 12790.385} C_VEL
LIN {X 0,Y 470.461,Z 596.746,A -85,B 0,C 180,E1 12788.064,E2 12788.064} C_VEL
LIN {X 0,Y 468.214,Z 592.444,A -85,B 0,C 180,E1 12785.269,E2 12785.269} C_VEL
LIN {X 0,Y 466.71,Z 588.723,A -85,B 0,C 180,E1 12781.473,E2 12781.473} C_VEL
LIN {X 0,Y 466.638,Z 588.149,A -85,B 0,C 180,E1 12780.737,E2 12780.737} C_VEL
LIN {X 0,Y 466.671,Z 588.355,A -85,B 0,C 180,E1 12778.404,E2 12778.404} C_VEL
LIN {X 0,Y 468.611,Z 593.243,A -85,B 0,C 180,E1 12773.63,E2 12773.63} C_VEL
LIN {X 0,Y 470.787,Z 597.565,A -85,B 0,C 180,E1 12771.081,E2 12771.081} C_VEL
LIN {X 0,Y 472.87,Z 601.713,A -85,B 0,C 180,E1 12769.214,E2 12769.214} C_VEL
LIN {X 0,Y 451.855,Z 807.705,A -85,B 0,C 180,E1 12766.241,E2 12766.241} C_VEL
LIN {X 0,Y 448.284,Z 831.594,A -85,B 0,C 180,E1 12765.852,E2 12765.852} C_VEL
LIN {X 0,Y 442.208,Z 860.791,A -85,B 0,C 180,E1 12765.245,E2 12765.245} C_VEL
LIN {X 0,Y 436.271,Z 883.295,A -85,B 0,C 180,E1 12764.64,E2 12764.64} C_VEL
LIN {X 0,Y 430.109,Z 903.208,A -85,B 0,C 180,E1 12763.996,E2 12763.996} C_VEL
LIN {X 0,Y 422.948,Z 923.418,A -85,B 0,C 180,E1 12763.221,E2 12763.221} C_VEL
LIN {X 0,Y 413.79,Z 946.186,A -85,B 0,C 180,E1 12762.182,E2 12762.182} C_VEL
LIN {X 0,Y 402.329,Z 970.904,A -85,B 0,C 180,E1 12760.798,E2 12760.798} C_VEL
LIN {X 0,Y 392.268,Z 990.25,A -85,B 0,C 180,E1 12759.508,E2 12759.508} C_VEL
LIN {X 0,Y 382.032,Z 1008.282,A -85,B 0,C 180,E1 12758.094,E2 12758.094} C_VEL
LIN {X 0,Y 370.899,Z 1026.369,A -85,B 0,C 180,E1 12756.428,E2 12756.428} C_VEL
LIN {X 0,Y 356.481,Z 1047.825,A -85,B 0,C 180,E1 12754.051,E2 12754.051} C_VEL
LIN {X 0,Y 343.951,Z 1064.915,A -85,B 0,C 180,E1 12751.74,E2 12751.74} C_VEL
LIN {X 0,Y 333.041,Z 1078.953,A -85,B 0,C 180,E1 12749.5,E2 12749.5} C_VEL
LIN {X 0,Y 322.007,Z 1092.455,A -85,B 0,C 180,E1 12746.968,E2 12746.968} C_VEL
LIN {X 0,Y 309.994,Z 1106.54,A -85,B 0,C 180,E1 12743.824,E2 12743.824} C_VEL
LIN {X 0,Y 295.963,Z 1122.268,A -85,B 0,C 180,E1 12739.475,E2 12739.475} C_VEL
LIN {X 0,Y 285.546,Z 1133.596,A -85,B 0,C 180,E1 12735.587,E2 12735.587} C_VEL
LIN {X 0,Y 276.785,Z 1143.098,A -85,B 0,C 180,E1 12731.658,E2 12731.658} C_VEL
LIN {X 0,Y 268.542,Z 1152.204,A -85,B 0,C 180,E1 12727.097,E2 12727.097} C_VEL
LIN {X 0,Y 259.919,Z 1162.14,A -85,B 0,C 180,E1 12720.772,E2 12720.772} C_VEL
LIN {X 0,Y 255.105,Z 1168.212,A -85,B 0,C 180,E1 12715.789,E2 12715.789} C_VEL
LIN {X 0,Y 251.827,Z 1172.921,A -85,B 0,C 180,E1 12710.937,E2 12710.937} C_VEL
